//Transport
//----------------------------------------P6015--------------------------------------------------------------
{attribute 'OPC.UA.DA' := '1'}
cfgP6015IntlksArry: ARRAY [0..15] OF ST_CfgEvents := [
   (Description := 'Exit PE/Downstream MTR status' , DeviceLabel := '' , OKState := TRUE),   //DeviceLabel: Exit PE downstream
   (Description := 'System Interlocks' , DeviceLabel := '', OKState := TRUE, StopCode := E_StopCodes.SystemStop),
   (),
   (Description := 'Powered Transfer Raised' , DeviceLabel := 'PX_1281', OKState := TRUE),
   11(())];
{attribute 'OPC.UA.DA' := '1'}
cfgP6015EvntsArry: ARRAY [0..15] OF ST_CfgEvents := [
   (Description := 'Jam Detected', DeviceLabel := '', LatchRequired := TRUE, OKState := FALSE, StopCode := E_StopCodes.ProductJam),   //DeviceLabel: Jam PE
   (),
   (Description := 'Disconnect', DeviceLabel := 'DS6015', OKState := TRUE, StopCode := E_StopCodes.DisconnectState),   //DeviceLabel: Motor Disconnect
   (Description := 'System Fault', DeviceLabel := 'System', OKState := TRUE, FaultWarn:= TRUE, StopCode := E_StopCodes.SystemStop),
   (Description := 'Fire Door Closed', DeviceLabel := 'PE_1231', OKState := TRUE, FaultWarn:= TRUE, StopCode := E_StopCodes.SystemStop),
   (Description := 'RIO1181 Comm Fault', DeviceLabel := 'RIO1181', OKState := TRUE, FaultWarn:= TRUE, StopCode := E_StopCodes.FieldIOFLT),
   (Description := 'Motor Faulted', DeviceLabel := 'P6015', OKState := FALSE, StopCode := E_StopCodes.MotorOL),
   9(())];
//----------------------------------------P6020--------------------------------------------------------------
{attribute 'OPC.UA.DA' := '1'}
cfgP6020IntlksArry: ARRAY [0..15] OF ST_CfgEvents := [
   (Description := 'Exit PE/Downstream MTR status' , DeviceLabel := '' , OKState := TRUE),   //DeviceLabel: Exit PE downstream
   (Description := 'System Interlocks' , DeviceLabel := '', OKState := TRUE, StopCode := E_StopCodes.SystemStop),
   (),
   13(())];
{attribute 'OPC.UA.DA' := '1'}
cfgP6020EvntsArry: ARRAY [0..15] OF ST_CfgEvents := [
   (Description := 'Jam Detected', DeviceLabel := '', LatchRequired := TRUE, OKState := FALSE, StopCode := E_StopCodes.ProductJam),   //DeviceLabel: Jam PE
   (),
   (Description := 'Disconnect', DeviceLabel := 'DS6020', OKState := TRUE, StopCode := E_StopCodes.DisconnectState),   //DeviceLabel: Motor Disconnect
   (Description := 'System Fault', DeviceLabel := 'System', OKState := TRUE, FaultWarn:= TRUE, StopCode := E_StopCodes.SystemStop),
   (Description := 'RIO16171 Comm Fault', DeviceLabel := 'RIO1181', OKState := TRUE, FaultWarn:= TRUE, StopCode := E_StopCodes.FieldIOFLT),
   (Description := 'Motor Faulted', DeviceLabel := 'P6020', OKState := FALSE, StopCode := E_StopCodes.MotorOL),
   10(())];
//----------------------------------------P6025--------------------------------------------------------------
{attribute 'OPC.UA.DA' := '1'}
cfgP6025IntlksArry: ARRAY [0..15] OF ST_CfgEvents := [
   (Description := 'Exit PE/Downstream MTR status' , DeviceLabel := '' , OKState := TRUE),   //DeviceLabel: Exit PE downstream
   (Description := 'System Interlocks' , DeviceLabel := '', OKState := TRUE, StopCode := E_StopCodes.SystemStop),
   (),
   13(())];
{attribute 'OPC.UA.DA' := '1'}
cfgP6025EvntsArry: ARRAY [0..15] OF ST_CfgEvents := [
   (Description := 'Jam Detected', DeviceLabel := '', LatchRequired := TRUE, OKState := FALSE, StopCode := E_StopCodes.ProductJam),   //DeviceLabel: Jam PE
   (),
   (Description := 'Disconnect', DeviceLabel := 'DS6025', OKState := TRUE, StopCode := E_StopCodes.DisconnectState),   //DeviceLabel: Motor Disconnect
   (Description := 'System Fault', DeviceLabel := 'System', OKState := TRUE, FaultWarn:= TRUE, StopCode := E_StopCodes.SystemStop),
   (Description := 'RIO4172 Comm Fault', DeviceLabel := 'RIO4172', OKState := TRUE, FaultWarn:= TRUE, StopCode := E_StopCodes.FieldIOFLT),
   (Description := 'Motor Faulted', DeviceLabel := 'P6025', OKState := FALSE, StopCode := E_StopCodes.MotorOL),
   10(())];
//----------------------------------------P6030--------------------------------------------------------------
{attribute 'OPC.UA.DA' := '1'}
cfgP6030IntlksArry: ARRAY [0..15] OF ST_CfgEvents := [
   (Description := 'Exit PE/Downstream MTR status' , DeviceLabel := '' , OKState := TRUE),   //DeviceLabel: Exit PE downstream
   (Description := 'System Interlocks' , DeviceLabel := '', OKState := TRUE, StopCode := E_StopCodes.SystemStop),
   (),
   12(())];
{attribute 'OPC.UA.DA' := '1'}
cfgP6030EvntsArry: ARRAY [0..15] OF ST_CfgEvents := [
   (Description := 'Jam Detected', DeviceLabel := '', LatchRequired := TRUE, OKState := FALSE, StopCode := E_StopCodes.ProductJam),   //DeviceLabel: Jam PE
   (),
   (Description := 'Disconnect', DeviceLabel := 'DS6030', OKState := TRUE, StopCode := E_StopCodes.DisconnectState),   //DeviceLabel: Motor Disconnect
   (Description := 'System Fault', DeviceLabel := 'System', OKState := TRUE, FaultWarn:= TRUE, StopCode := E_StopCodes.SystemStop),
   (Description := 'RIO4172 Comm Fault', DeviceLabel := 'RIO4172', OKState := TRUE, FaultWarn:= TRUE, StopCode := E_StopCodes.FieldIOFLT),
   (Description := 'Motor Faulted', DeviceLabel := 'P6030', OKState := FALSE, StopCode := E_StopCodes.MotorOL),
   10(())];
//----------------------------------------P6035--------------------------------------------------------------
{attribute 'OPC.UA.DA' := '1'}
cfgP6035IntlksArry: ARRAY [0..15] OF ST_CfgEvents := [
   (Description := 'Exit PE/Downstream MTR status' , DeviceLabel := '' , OKState := TRUE),   //DeviceLabel: Exit PE downstream
   (Description := 'System Interlocks' , DeviceLabel := '', OKState := TRUE, StopCode := E_StopCodes.SystemStop),
   (),
   12(())];
{attribute 'OPC.UA.DA' := '1'}
cfgP6035EvntsArry: ARRAY [0..15] OF ST_CfgEvents := [
   (Description := 'Jam Detected', DeviceLabel := '', LatchRequired := TRUE, OKState := FALSE, StopCode := E_StopCodes.ProductJam),   //DeviceLabel: Jam PE
   (),
   (Description := 'Disconnect', DeviceLabel := 'DS6035', OKState := TRUE, StopCode := E_StopCodes.DisconnectState),   //DeviceLabel: Motor Disconnect
   (Description := 'System Fault', DeviceLabel := 'System', OKState := TRUE, FaultWarn:= TRUE, StopCode := E_StopCodes.SystemStop),
   (Description := 'RIO4172 Comm Fault', DeviceLabel := 'RIO4172', OKState := TRUE, FaultWarn:= TRUE, StopCode := E_StopCodes.FieldIOFLT),
   (Description := 'Motor Faulted', DeviceLabel := 'P6035', OKState := FALSE, StopCode := E_StopCodes.MotorOL),
   10(())];
//Spiral
//----------------------------------------P6045--------------------------------------------------------------
{attribute 'OPC.UA.DA' := '1'}
cfgP6045IntlksArry: ARRAY [0..15] OF ST_CfgEvents := [
   (Description := 'Exit PE/Downstream MTR status' , DeviceLabel := '' , OKState := TRUE),   //DeviceLabel: Exit PE downstream
   (Description := 'System Interlocks' , DeviceLabel := '', OKState := TRUE, StopCode := E_StopCodes.SystemStop),
   (),
   12(())];
{attribute 'OPC.UA.DA' := '1'}
cfgP6045EvntsArry: ARRAY [0..15] OF ST_CfgEvents := [
   (Description := 'Jam Detected', DeviceLabel := '', LatchRequired := TRUE, OKState := FALSE, StopCode := E_StopCodes.ProductJam),   //DeviceLabel: Jam PE
   (),
   (Description := 'Disconnect', DeviceLabel := 'DS6045', OKState := TRUE, StopCode := E_StopCodes.DisconnectState),   //DeviceLabel: Motor Disconnect
   (Description := 'System Fault', DeviceLabel := 'System', OKState := TRUE, FaultWarn:= TRUE, StopCode := E_StopCodes.SystemStop),
   (Description := 'RIO4172 Comm Fault', DeviceLabel := 'RIO4172', OKState := TRUE, FaultWarn:= TRUE, StopCode := E_StopCodes.FieldIOFLT),
   (Description := 'VFD State Not OK', DeviceLabel := 'P6045', OKState := TRUE, StopCode := E_StopCodes.VFD_Fault),
   10(())];
//Sorter
//----------------------------------------P6040--------------------------------------------------------------
{attribute 'OPC.UA.DA' := '1'}
cfgP6040IntlksArry: ARRAY [0..15] OF ST_CfgEvents := [
   (Description := 'Exit PE/Downstream MTR status' , DeviceLabel := '' , OKState := TRUE),   //DeviceLabel: Exit PE downstream
   (Description := 'System Interlocks' , DeviceLabel := '', OKState := TRUE, StopCode := E_StopCodes.SystemStop),
   (Description := 'GR6040-01 Auto', DeviceLabel := 'GR6040-01', OKState := TRUE, StopCode := E_StopCodes.DeviceNoInAuto),
   (Description := 'GR6040-02 Auto', DeviceLabel := 'GR6040-02', OKState := TRUE, StopCode := E_StopCodes.DeviceNoInAuto),
   (Description := 'PI6040-01 Auto', DeviceLabel := 'PI6040-01', OKState := TRUE, StopCode := E_StopCodes.DeviceNoInAuto),
   (Description := 'PU6040-01 Auto', DeviceLabel := 'PU6040-01', OKState := TRUE, StopCode := E_StopCodes.DeviceNoInAuto),
   (Description := 'PU6040-02 Auto', DeviceLabel := 'PU6040-02', OKState := TRUE, StopCode := E_StopCodes.DeviceNoInAuto),
   (Description := 'PU6040-03 Auto', DeviceLabel := 'PU6040-03', OKState := TRUE, StopCode := E_StopCodes.DeviceNoInAuto),
   (Description := 'PU6040-04 Auto', DeviceLabel := 'PU6040-04', OKState := TRUE, StopCode := E_StopCodes.DeviceNoInAuto),
   (Description := 'Motor Faulted', DeviceLabel := 'P6030', OKState := FALSE, StopCode := E_StopCodes.MotorOL),
   6(())];
{attribute 'OPC.UA.DA' := '1'}
cfgP6040EvntsArry: ARRAY [0..15] OF ST_CfgEvents := [
   (Description := 'Jam Detected', DeviceLabel := '', LatchRequired := TRUE, OKState := FALSE, StopCode := E_StopCodes.ProductJam),   //DeviceLabel: Jam PE
   (),
   (Description := 'Disconnect', DeviceLabel := 'DS6040', OKState := TRUE, StopCode := E_StopCodes.DisconnectState),   //DeviceLabel: Motor Disconnect
   (Description := 'System Fault', DeviceLabel := 'System', OKState := TRUE, FaultWarn:= TRUE, StopCode := E_StopCodes.SystemStop),
   (Description := 'RIO6171 Comm Fault', DeviceLabel := 'RIO6171', OKState := TRUE, FaultWarn:= TRUE, StopCode := E_StopCodes.FieldIOFLT),
   (Description := 'RIO7161 Comm Fault', DeviceLabel := 'RIO7161', OKState := TRUE, FaultWarn:= TRUE, StopCode := E_StopCodes.FieldIOFLT),
   (Description := 'RIO8181 Comm Fault', DeviceLabel := 'RIO8081', OKState := TRUE, FaultWarn:= TRUE, StopCode := E_StopCodes.FieldIOFLT),
   (Description := 'Motor Faulted', DeviceLabel := 'P6030', OKState := FALSE, StopCode := E_StopCodes.MotorOL),
   8(())];
//Conveyors Outgoing 7000 (Orange line)
//Loading Zone
//----------------------------------------P7004--------------------------------------------------------------
{attribute 'OPC.UA.DA' := '1'}
cfgP7004IntlksArry: ARRAY [0..15] OF ST_CfgEvents := [
   (Description := 'Exit PE/Downstream MTR status' , DeviceLabel := '' , OKState := TRUE),   //DeviceLabel: Exit PE downstream
   (Description := 'System Interlocks' , DeviceLabel := '', OKState := TRUE, StopCode := E_StopCodes.SystemStop),
   (),
   12(())];
{attribute 'OPC.UA.DA' := '1'}
cfgP7004EvntsArry: ARRAY [0..15] OF ST_CfgEvents := [
   (Description := 'Jam Detected', DeviceLabel := '', LatchRequired := TRUE, OKState := FALSE, StopCode := E_StopCodes.ProductJam),   //DeviceLabel: Jam PE
   (),
   (Description := 'Disconnect', DeviceLabel := 'DS7004', OKState := TRUE, StopCode := E_StopCodes.DisconnectState),   //DeviceLabel: Motor Disconnect
   (Description := 'System Fault', DeviceLabel := 'System', OKState := TRUE, FaultWarn:= TRUE, StopCode := E_StopCodes.SystemStop),
   (Description := 'Height Check', DeviceLabel := 'PE_12261', OKState := TRUE, FaultWarn:= TRUE, StopCode := E_StopCodes.OverHeightFLT),
   (Description := 'RIO12171 Comm Fault', DeviceLabel := 'RIO12171', OKState := TRUE, FaultWarn:= TRUE, StopCode := E_StopCodes.FieldIOFLT),
   (Description := 'Motor Faulted', DeviceLabel := 'P6030', OKState := FALSE, StopCode := E_StopCodes.MotorOL),
   9(())];
//Spiral
//----------------------------------------P7005--------------------------------------------------------------
{attribute 'OPC.UA.DA' := '1'}
cfgP7005IntlksArry: ARRAY [0..15] OF ST_CfgEvents := [
   (Description := 'Exit PE/Downstream MTR status' , DeviceLabel := '' , OKState := TRUE),   //DeviceLabel: Exit PE downstream
   (Description := 'System Interlocks' , DeviceLabel := '', OKState := TRUE, StopCode := E_StopCodes.SystemStop),
   (),
   12(())];
{attribute 'OPC.UA.DA' := '1'}
cfgP7005EvntsArry: ARRAY [0..15] OF ST_CfgEvents := [
   (Description := 'Jam Detected', DeviceLabel := '', LatchRequired := TRUE, OKState := FALSE, StopCode := E_StopCodes.ProductJam),   //DeviceLabel: Jam PE
   (),
   (Description := 'Disconnect', DeviceLabel := 'DS7005', OKState := TRUE, StopCode := E_StopCodes.DisconnectState),   //DeviceLabel: Motor Disconnect
   (Description := 'System Fault', DeviceLabel := 'System', OKState := TRUE, FaultWarn:= TRUE, StopCode := E_StopCodes.SystemStop),
   (Description := 'RIO12171 Comm Fault', DeviceLabel := 'RIO12171', OKState := TRUE, FaultWarn:= TRUE, StopCode := E_StopCodes.FieldIOFLT),
   (Description := 'VFD State Not OK', DeviceLabel := 'P7005', OKState := TRUE, StopCode := E_StopCodes.VFD_Fault),
   10(())];
//Transport
//----------------------------------------P7010--------------------------------------------------------------
{attribute 'OPC.UA.DA' := '1'}
cfgP7010IntlksArry: ARRAY [0..15] OF ST_CfgEvents := [
   (Description := 'Exit PE/Downstream MTR status' , DeviceLabel := '' , OKState := TRUE),   //DeviceLabel: Exit PE downstream
   (Description := 'System Interlocks' , DeviceLabel := '', OKState := TRUE, StopCode := E_StopCodes.SystemStop),
   (),
   12(())];
{attribute 'OPC.UA.DA' := '1'}
cfgP7010EvntsArry: ARRAY [0..15] OF ST_CfgEvents := [
   (Description := 'Jam Detected', DeviceLabel := '', LatchRequired := TRUE, OKState := FALSE, StopCode := E_StopCodes.ProductJam),   //DeviceLabel: Jam PE
   (),
   (Description := 'Disconnect', DeviceLabel := '', OKState := TRUE, StopCode := E_StopCodes.DisconnectState),   //DeviceLabel: Motor Disconnect
   (Description := 'System Fault', DeviceLabel := 'System', OKState := TRUE, FaultWarn:= TRUE, StopCode := E_StopCodes.SystemStop),
   (Description := 'RIO12171 Comm Fault', DeviceLabel := 'RIO12171', OKState := TRUE, FaultWarn:= TRUE, StopCode := E_StopCodes.FieldIOFLT),
   (Description := 'Motor Faulted', DeviceLabel := 'P7010', OKState := FALSE, StopCode := E_StopCodes.MotorOL),
   10(())];
//----------------------------------------P7015--------------------------------------------------------------
{attribute 'OPC.UA.DA' := '1'}
cfgP7015IntlksArry: ARRAY [0..15] OF ST_CfgEvents := [
   (Description := 'Exit PE/Downstream MTR status' , DeviceLabel := '' , OKState := TRUE),   //DeviceLabel: Exit PE downstream
   (Description := 'System Interlocks' , DeviceLabel := '', OKState := TRUE, StopCode := E_StopCodes.SystemStop),
   (),
   12(())];
{attribute 'OPC.UA.DA' := '1'}
cfgP7015EvntsArry: ARRAY [0..15] OF ST_CfgEvents := [
   (Description := 'Jam Detected', DeviceLabel := '', LatchRequired := TRUE, OKState := FALSE, StopCode := E_StopCodes.ProductJam),   //DeviceLabel: Jam PE
   (),
   (Description := 'Disconnect', DeviceLabel := '', OKState := TRUE, StopCode := E_StopCodes.DisconnectState),   //DeviceLabel: Motor Disconnect
   (Description := 'System Fault', DeviceLabel := 'System', OKState := TRUE, FaultWarn:= TRUE, StopCode := E_StopCodes.SystemStop),
   (Description := 'RIO15181 Comm Fault', DeviceLabel := 'RIO15181', OKState := TRUE, FaultWarn:= TRUE, StopCode := E_StopCodes.FieldIOFLT),
   (Description := 'Motor Faulted', DeviceLabel := 'P7015', OKState := FALSE, StopCode := E_StopCodes.MotorOL),
   10(())];
//----------------------------------------P7020--------------------------------------------------------------
{attribute 'OPC.UA.DA' := '1'}
cfgP7020IntlksArry: ARRAY [0..15] OF ST_CfgEvents := [
   (Description := 'Exit PE/Downstream MTR status' , DeviceLabel := '' , OKState := TRUE),   //DeviceLabel: Exit PE downstream
   (Description := 'System Interlocks' , DeviceLabel := '', OKState := TRUE, StopCode := E_StopCodes.SystemStop),
   (),
   12(())];
{attribute 'OPC.UA.DA' := '1'}
cfgP7020EvntsArry: ARRAY [0..15] OF ST_CfgEvents := [
   (Description := 'Jam Detected', DeviceLabel := '', LatchRequired := TRUE, OKState := FALSE, StopCode := E_StopCodes.ProductJam),   //DeviceLabel: Jam PE
   (),
   (Description := 'Disconnect', DeviceLabel := '', OKState := TRUE, StopCode := E_StopCodes.DisconnectState),   //DeviceLabel: Motor Disconnect
   (Description := 'System Fault', DeviceLabel := 'System', OKState := TRUE, FaultWarn:= TRUE, StopCode := E_StopCodes.SystemStop),
   (Description := 'RIO15181 Comm Fault', DeviceLabel := 'RIO15181', OKState := TRUE, FaultWarn:= TRUE, StopCode := E_StopCodes.FieldIOFLT),
   (Description := 'Motor Faulted', DeviceLabel := 'P7020', OKState := FALSE, StopCode := E_StopCodes.MotorRunTO),
   10(())];
//----------------------------------------P7025--------------------------------------------------------------
{attribute 'OPC.UA.DA' := '1'}
cfgP7025IntlksArry: ARRAY [0..15] OF ST_CfgEvents := [
   (Description := 'Exit PE/Downstream MTR status' , DeviceLabel := '' , OKState := TRUE),   //DeviceLabel: Exit PE downstream
   (Description := 'System Interlocks' , DeviceLabel := '', OKState := TRUE, StopCode := E_StopCodes.SystemStop),
   (),
   12(())];
{attribute 'OPC.UA.DA' := '1'}
cfgP7025EvntsArry: ARRAY [0..15] OF ST_CfgEvents := [
   (Description := 'Jam Detected', DeviceLabel := '', LatchRequired := TRUE, OKState := FALSE, StopCode := E_StopCodes.ProductJam),   //DeviceLabel: Jam PE
   (),
   (Description := 'Disconnect', DeviceLabel := '', OKState := TRUE, StopCode := E_StopCodes.DisconnectState),   //DeviceLabel: Motor Disconnect
   (Description := 'System Fault', DeviceLabel := 'System', OKState := TRUE, FaultWarn:= TRUE, StopCode := E_StopCodes.SystemStop),
   (Description := 'RIO15181 Comm Fault', DeviceLabel := 'RIO15181', OKState := TRUE, FaultWarn:= TRUE, StopCode := E_StopCodes.FieldIOFLT),
   (Description := 'Motor Faulted', DeviceLabel := 'P7025', OKState := FALSE, StopCode := E_StopCodes.MotorOL),
   10(())];
//----------------------------------------P7030--------------------------------------------------------------
{attribute 'OPC.UA.DA' := '1'}
cfgP7030IntlksArry: ARRAY [0..15] OF ST_CfgEvents := [
   (Description := 'Exit PE/Downstream MTR status' , DeviceLabel := '' , OKState := TRUE),   //DeviceLabel: Exit PE downstream
   (Description := 'System Interlocks' , DeviceLabel := '', OKState := TRUE, StopCode := E_StopCodes.SystemStop),
   (),
   12(())];
{attribute 'OPC.UA.DA' := '1'}
cfgP7030EvntsArry: ARRAY [0..15] OF ST_CfgEvents := [
   (Description := 'Jam Detected', DeviceLabel := '', LatchRequired := TRUE, OKState := FALSE, StopCode := E_StopCodes.ProductJam),   //DeviceLabel: Jam PE
   (),
   (Description := 'Disconnect', DeviceLabel := '', OKState := TRUE, StopCode := E_StopCodes.DisconnectState),   //DeviceLabel: Motor Disconnect
   (Description := 'System Fault', DeviceLabel := 'System', OKState := TRUE, FaultWarn:= TRUE, StopCode := E_StopCodes.SystemStop),
   (Description := 'RIO16171 Comm Fault', DeviceLabel := 'RIO16171', OKState := TRUE, FaultWarn:= TRUE, StopCode := E_StopCodes.FieldIOFLT),
   (Description := 'Motor Faulted', DeviceLabel := 'P7030', OKState := FALSE, StopCode := E_StopCodes.MotorOL),
   10(())];
//----------------------------------------P7035--------------------------------------------------------------
{attribute 'OPC.UA.DA' := '1'}
cfgP7035IntlksArry: ARRAY [0..15] OF ST_CfgEvents := [
   (Description := 'Exit PE/Downstream MTR status' , DeviceLabel := '' , OKState := TRUE),   //DeviceLabel: Exit PE downstream
   (Description := 'System Interlocks' , DeviceLabel := '', OKState := TRUE, StopCode := E_StopCodes.SystemStop),
   (),
   (Description := 'Powered Transfer Raised' , DeviceLabel := 'PX_16231', OKState := TRUE),
   12(())];
{attribute 'OPC.UA.DA' := '1'}
cfgP7035EvntsArry: ARRAY [0..15] OF ST_CfgEvents := [
   (Description := 'Jam Detected', DeviceLabel := '', LatchRequired := TRUE, OKState := FALSE, StopCode := E_StopCodes.ProductJam),   //DeviceLabel: Jam PE
   (),
   (Description := 'Disconnect', DeviceLabel := '', OKState := TRUE, StopCode := E_StopCodes.DisconnectState),   //DeviceLabel: Motor Disconnect
   (Description := 'System Fault', DeviceLabel := 'System', OKState := TRUE, FaultWarn:= TRUE, StopCode := E_StopCodes.SystemStop),
   (Description := 'Fire Door Closed', DeviceLabel := 'PE_16181', OKState := TRUE, FaultWarn:= TRUE, StopCode := E_StopCodes.SystemStop),
   (Description := 'RIO16171 Comm Fault', DeviceLabel := 'RIO16171', OKState := TRUE, FaultWarn:= TRUE, StopCode := E_StopCodes.FieldIOFLT),
   (Description := 'Motor Faulted', DeviceLabel := 'P7035', OKState := FALSE, StopCode := E_StopCodes.MotorOL),
   9(())];
//Spiral
//----------------------------------------P7040--------------------------------------------------------------
{attribute 'OPC.UA.DA' := '1'}
cfgP7040IntlksArry: ARRAY [0..15] OF ST_CfgEvents := [
   (Description := 'Exit PE/Downstream MTR status' , DeviceLabel := '' , OKState := TRUE),   //DeviceLabel: Exit PE downstream
   (Description := 'System Interlocks' , DeviceLabel := '', OKState := TRUE, StopCode := E_StopCodes.SystemStop),
   (),
   13(())];
{attribute 'OPC.UA.DA' := '1'}
cfgP7040EvntsArry: ARRAY [0..15] OF ST_CfgEvents := [
   (Description := 'Jam Detected', DeviceLabel := '', LatchRequired := TRUE, OKState := FALSE, StopCode := E_StopCodes.ProductJam),   //DeviceLabel: Jam PE
   (),
   (Description := 'Disconnect', DeviceLabel := '', OKState := TRUE, StopCode := E_StopCodes.DisconnectState),   //DeviceLabel: Motor Disconnect
   (Description := 'System Fault', DeviceLabel := 'System', OKState := TRUE, FaultWarn:= TRUE, StopCode := E_StopCodes.SystemStop),
   (Description := 'RIO16171 Comm Fault', DeviceLabel := 'RIO16171', OKState := TRUE, FaultWarn:= TRUE, StopCode := E_StopCodes.FieldIOFLT),
   (Description := 'VFD State Not OK', DeviceLabel := 'P7040', OKState := TRUE, StopCode := E_StopCodes.VFD_Fault),
   10(())];

//Transport
//----------------------------------------P7045--------------------------------------------------------------
{attribute 'OPC.UA.DA' := '1'}
cfgP7045IntlksArry: ARRAY [0..15] OF ST_CfgEvents := [
   (Description := 'Exit PE/Downstream MTR status' , DeviceLabel := '' , OKState := TRUE),   //DeviceLabel: Exit PE downstream
   (Description := 'System Interlocks' , DeviceLabel := '', OKState := TRUE, StopCode := E_StopCodes.SystemStop),
   (),
   13(())];
{attribute 'OPC.UA.DA' := '1'}
cfgP7045EvntsArry: ARRAY [0..15] OF ST_CfgEvents := [
   (Description := 'Jam Detected', DeviceLabel := '', LatchRequired := TRUE, OKState := FALSE, StopCode := E_StopCodes.ProductJam),   //DeviceLabel: Jam PE
   (),
   (Description := 'Disconnect', DeviceLabel := '', OKState := TRUE, StopCode := E_StopCodes.DisconnectState),   //DeviceLabel: Motor Disconnect
   (Description := 'System Fault', DeviceLabel := 'System', OKState := TRUE, FaultWarn:= TRUE, StopCode := E_StopCodes.SystemStop),
   (Description := 'Fire Door Closed', DeviceLabel := 'PE_16181', OKState := TRUE, FaultWarn:= TRUE, StopCode := E_StopCodes.SystemStop),
   (Description := 'RIO16171 Comm Fault', DeviceLabel := 'RIO16171', OKState := TRUE, FaultWarn:= TRUE, StopCode := E_StopCodes.FieldIOFLT),
   (Description := 'Motor Faulted', DeviceLabel := 'P7045', OKState := FALSE, StopCode := E_StopCodes.MotorOL),
   9(())];			
END_VAR

ResetAllDrives:=System.Cnvyr_Reset;

//----------------------------------------P6005--------------------------------------------------------------
P6005_StatePB.AutoPB := System.Cnvyr_Auto;
P6005_StatePB.ManPB := System.Cnvyr_Manual;
P6005_StatePB.ResetPB := System.Cnvyr_Reset;
P6005_StatePB.OfflinePB := System.Cnvyr_Offline;
P6005SleepWakeTrig[1] := PhotoEyes.PE_1232.Out;
P6005SleepWakeTrig[2] := GVL_IO.From205_P3130_SendingProduct;		// Belive this will be an EAP photoeye from 3rd floor

GVL_IO.To205_P6005_IsRunning:= P6005_Status.Sts_IsRunning;

// Initialize the Equipment Type
P6005_Status.Sts_EquipmentState.EquipType := E_EquipType.Conveyor;

// Interlocks
//P6005.In_EquipIntlks.2:=  

//Events
  P6005.In_EquipEvents.2:= GVL_IO.DS_P6005;
  P6005.In_EquipEvents.3:= System.SysEventsAllOk;
  P6005.In_EquipEvents.4:= Photoeyes.PE_1231.Out; //Goes low when door drops
  P6005.In_EquipEvents.5:= NOT CommStatus.RIO1181_CommFault.Out;
  P6005.In_EquipEvents.6:= NOT GVL_IO.P6005_Faulted;

// Function Call
P6005(
   In_p_EquipStatePB:= P6005_StatePB,
   In_P_ConvReqRun:= TRUE,
   In_ConvDwnStrmMtrStatus:= P6010_VFD.IsRunning,
   In_ConvCrntExitPhotoEye:= Photoeyes.PE_1232.Out,
   In_SimActive:= System.Sys_SimActive,
   In_EquipInit:= GVL_IO.INIT,
   In_WakeSlpTrigArry:= P6005SleepWakeTrig,
   Cfg_EquipIndex := GVL_EquipArrays.nEquipIndex,
   Cfg_EquipLabel := cfgP6005Label,
   Cfg_EquipDefState:= System.ConvDefaultState,
   Cfg_EquipIntlksArry:= cfgP6005IntlksArry,
   Cfg_EquipEvntsArry:= cfgP6005EvntsArry,
   cfg_JamDetectTime:= cfgP6005JamDetectTime,
   Cfg_UseSleepTmr := TRUE,
   Cfg_UseStartUpDelay := TRUE,
   Cfg_StartUpDelayTime := T#500MS,
   Cfg_SleepWaitTime:= cfgP6005SleepTime,
   Sts_EquipState := P6005_Status,
   Out_ConvCrntMtr => GVL_IO.P6005_RUN);

P6005_Status.Sts_IsRunning := GVL_IO.P6005_RUN;
//----------------------------------------P6010--------------------------------------------------------------
P6010_StatePB.AutoPB := System.Cnvyr_Auto;
P6010_StatePB.ManPB := System.Cnvyr_Manual;
P6010_StatePB.ResetPB := System.Cnvyr_Reset;
P6010_StatePB.OfflinePB := System.Cnvyr_Offline;
P6010SleepWakeTrig[1] := PhotoEyes.PE_1232.Out_OffFltrd;
P6010SleepWakeTrig[5] := P6005SleepWakeTrig[1]
						OR P6005SleepWakeTrig[2]
						OR P6005SleepWakeTrig[3]
						OR P6005SleepWakeTrig[4]
						OR P6005SleepWakeTrig[5];
// ADD an EAP photoeye from 3rd floor

// Initialize the Equipment Type
P6010_Status.Sts_EquipmentState.EquipType := E_EquipType.Conveyor;

// Interlocks
 // P6010.In_EquipIntlks.2:= 
//Events
  P6010.In_EquipEvents.2:= GVL_IO.DS_P6010;
  P6010.In_EquipEvents.3:= System.SysEventsAllOk;
  P6010.In_EquipEvents.4:= NOT CommStatus.RIO1181_CommFault.Out;
  P6010.In_EquipEvents.5:= NOT P6010_VFD.IsFaulted;

// Function Call
P6010(
   In_p_EquipStatePB:= P6010_StatePB,
   In_P_ConvReqRun:= TRUE,
   In_ConvDwnStrmMtrStatus:= P6015_Status.Sts_IsRunning,
   In_ConvCrntExitPhotoEye:= Photoeyes.PE_1162.Out,
   In_SimActive:= System.Sys_SimActive,
   In_EquipInit:= GVL_IO.INIT,
   In_WakeSlpTrigArry:= P6010SleepWakeTrig,
   Cfg_EquipIndex := GVL_EquipArrays.nEquipIndex,
   Cfg_EquipLabel := cfgP6010Label,
   Cfg_EquipDefState:= System.ConvDefaultState,
   Cfg_EquipIntlksArry:= cfgP6010IntlksArry,
   Cfg_EquipEvntsArry:= cfgP6010EvntsArry,
   cfg_JamDetectTime:= cfgP6010JamDetectTime,
   Cfg_UseSleepTmr := TRUE,
   Cfg_UseStartUpDelay := TRUE,
   Cfg_StartUpDelayTime := T#500MS,
   Cfg_SleepWaitTime:= cfgP6010SleepTime,
   Sts_EquipState := P6010_Status);

//Motor Control
P6010_VFD(
   RunVelocity := DefaultVelocity,
   VelocityThreshold := DefaultVelocityThreshold,
   Reset := ResetAllDrives,
   RunRequest := (P6010.Out_ConvCrntMtr OR Test_VFD_P6010));
P6010_Status.Sts_IsRunning := P6010_VFD.IsRunning;

//----------------------------------------P6015--------------------------------------------------------------
P6015_StatePB.AutoPB := System.Cnvyr_Auto;
P6015_StatePB.ManPB := System.Cnvyr_Manual;
P6015_StatePB.ResetPB := System.Cnvyr_Reset;
P6015_StatePB.OfflinePB := System.Cnvyr_Offline;
P6015SleepWakeTrig[1] := PhotoEyes.PE_1162.Out_OffFltrd;
P6015SleepWakeTrig[2] :=  PhotoEyes.PE_1232.Out_OffFltrd;

// Initialize the Equipment Type
P6015_Status.Sts_EquipmentState.EquipType := E_EquipType.Conveyor;

// Interlocks
  P6015.In_EquipIntlks.3:= ProxSensors.PX_1281_Extended.Out; //Powered Transfer Raised 
//Events
  P6015.In_EquipEvents.2:= GVL_IO.DS_P6015;
  P6015.In_EquipEvents.3:= System.SysEventsAllOk;
  P6015.In_EquipEvents.4:= Photoeyes.PE_1231.Out; //Goes low when door drops
  P6015.In_EquipEvents.5:= NOT CommStatus.RIO1181_CommFault.Out;
  P6015.In_EquipEvents.6:= NOT GVL_IO.P6015_Faulted;

// Function Call
P6015(
   In_p_EquipStatePB:= P6015_StatePB,
   In_P_ConvReqRun:= TRUE,
   In_ConvDwnStrmMtrStatus:= P6020_Status.Sts_IsRunning,
   In_ConvCrntExitPhotoEye:= Photoeyes.PE_1081.Out,
   In_SimActive:= System.Sys_SimActive,
   In_EquipInit:= GVL_IO.INIT,
   In_WakeSlpTrigArry:= P6015SleepWakeTrig,
   Cfg_EquipIndex := GVL_EquipArrays.nEquipIndex,
   Cfg_EquipLabel := cfgP6015Label,
   Cfg_EquipDefState:= System.ConvDefaultState,
   Cfg_EquipIntlksArry:= cfgP6015IntlksArry,
   Cfg_EquipEvntsArry:= cfgP6015EvntsArry,
   cfg_JamDetectTime:= cfgP6015JamDetectTime,
   Cfg_UseSleepTmr := TRUE,
   Cfg_UseStartUpDelay := TRUE,
   Cfg_StartUpDelayTime := T#500MS,
   Cfg_SleepWaitTime:= cfgP6015SleepTime,
   Sts_EquipState := P6015_Status,
   Out_ConvCrntMtr => GVL_IO.P6015_RUN);

P6015_Status.Sts_IsRunning := GVL_IO.P6015_RUN;
//----------------------------------------P6020--------------------------------------------------------------
P6020_StatePB.AutoPB := System.Cnvyr_Auto;
P6020_StatePB.ManPB := System.Cnvyr_Manual;
P6020_StatePB.ResetPB := System.Cnvyr_Reset;
P6020_StatePB.OfflinePB := System.Cnvyr_Offline;
P6020SleepWakeTrig[1] := PhotoEyes.PE_1081.Out_OffFltrd;
P6020SleepWakeTrig[2] := PhotoEyes.PE_1162.Out_OffFltrd;

// Initialize the Equipment Type
P6020_Status.Sts_EquipmentState.EquipType := E_EquipType.Conveyor;

// Interlocks
 // P6020.In_EquipIntlks.2:=
//Events
  P6020.In_EquipEvents.2:= GVL_IO.DS_P6020;
  P6020.In_EquipEvents.3:= System.SysEventsAllOk;
  P6020.In_EquipEvents.4:= NOT CommStatus.RIO1181_CommFault.Out;
  P6020.In_EquipEvents.5:= NOT GVL_IO.P6020_Faulted;

// Function Call
P6020(
   In_p_EquipStatePB:= P6020_StatePB,
   In_P_ConvReqRun:= TRUE,
   In_ConvDwnStrmMtrStatus:= P6025_Status.Sts_IsRunning,
   In_ConvCrntExitPhotoEye:= Photoeyes.PE_1161.Out,
   In_SimActive:= System.Sys_SimActive,
   In_EquipInit:= GVL_IO.INIT,
   In_WakeSlpTrigArry:= P6020SleepWakeTrig,
   Cfg_EquipIndex := GVL_EquipArrays.nEquipIndex,
   Cfg_EquipLabel := cfgP6020Label,
   Cfg_EquipDefState:= System.ConvDefaultState,
   Cfg_EquipIntlksArry:= cfgP6020IntlksArry,
   Cfg_EquipEvntsArry:= cfgP6020EvntsArry,
   cfg_JamDetectTime:= cfgP6020JamDetectTime,
   Cfg_UseSleepTmr := TRUE,
   Cfg_UseStartUpDelay := TRUE,
   Cfg_StartUpDelayTime := T#500MS,
   Cfg_SleepWaitTime:= cfgP6020SleepTime,
   Sts_EquipState := P6020_Status,
   Out_ConvCrntMtr => GVL_IO.P6020_RUN);

P6020_Status.Sts_IsRunning := GVL_IO.P6020_RUN;
//----------------------------------------P6025--------------------------------------------------------------
P6025_StatePB.AutoPB := System.Cnvyr_Auto;
P6025_StatePB.ManPB := System.Cnvyr_Manual;
P6025_StatePB.ResetPB := System.Cnvyr_Reset;
P6025_StatePB.OfflinePB := System.Cnvyr_Offline;
P6025SleepWakeTrig[1] := PhotoEyes.PE_1161.Out_OffFltrd;
P6025SleepWakeTrig[2] := PhotoEyes.PE_1081.Out_OffFltrd;

// Initialize the Equipment Type
P6025_Status.Sts_EquipmentState.EquipType := E_EquipType.Conveyor;

// Interlocks
//  P6025.In_EquipIntlks.2:= 
//Events
  P6025.In_EquipEvents.2:= GVL_IO.DS_P6025;
  P6025.In_EquipEvents.3:= System.SysEventsAllOk;
  P6025.In_EquipEvents.4:= NOT CommStatus.RIO4172_CommFault.Out;
  P6025.In_EquipEvents.5:= NOT GVL_IO.P6025_Faulted;

// Function Call
P6025(
   In_p_EquipStatePB:= P6025_StatePB,
   In_P_ConvReqRun:= TRUE,
   In_ConvDwnStrmMtrStatus:= P6030_Status.Sts_IsRunning,
   In_ConvCrntExitPhotoEye:= Photoeyes.PE_4121.Out,
   In_SimActive:= System.Sys_SimActive,
   In_EquipInit:= GVL_IO.INIT,
   In_WakeSlpTrigArry:= P6025SleepWakeTrig,
   Cfg_EquipIndex := GVL_EquipArrays.nEquipIndex,
   Cfg_EquipLabel := cfgP6025Label,
   Cfg_EquipDefState:= System.ConvDefaultState,
   Cfg_EquipIntlksArry:= cfgP6025IntlksArry,
   Cfg_EquipEvntsArry:= cfgP6025EvntsArry,
   cfg_JamDetectTime:= cfgP6025JamDetectTime,
   Cfg_UseSleepTmr := TRUE,
   Cfg_UseStartUpDelay := TRUE,
   Cfg_StartUpDelayTime := T#500MS,
   Cfg_SleepWaitTime:= cfgP6025SleepTime,
   Sts_EquipState := P6025_Status,
   Out_ConvCrntMtr => GVL_IO.P6025_RUN);

P6025_Status.Sts_IsRunning := GVL_IO.P6025_RUN;
//----------------------------------------P6030--------------------------------------------------------------
P6030_StatePB.AutoPB := System.Cnvyr_Auto;
P6030_StatePB.ManPB := System.Cnvyr_Manual;
P6030_StatePB.ResetPB := System.Cnvyr_Reset;
P6030_StatePB.OfflinePB := System.Cnvyr_Offline;
P6030SleepWakeTrig[1] := PhotoEyes.PE_4121.Out_OffFltrd;
P6030SleepWakeTrig[2] := PhotoEyes.PE_1161.Out_OffFltrd;

// Initialize the Equipment Type
P6030_Status.Sts_EquipmentState.EquipType := E_EquipType.Conveyor;

// Interlocks
// P6030.In_EquipIntlks.2:= 
//Events
  P6030.In_EquipEvents.2:= GVL_IO.DS_P6030;
  P6030.In_EquipEvents.3:= System.SysEventsAllOk;
  P6030.In_EquipEvents.4:= NOT CommStatus.RIO4172_CommFault.Out;
  P6030.In_EquipEvents.5:= NOT GVL_IO.P6030_Faulted;

// Function Call
P6030(
   In_p_EquipStatePB:= P6030_StatePB,
   In_P_ConvReqRun:= TRUE,
   In_ConvDwnStrmMtrStatus:= P6035_Status.Sts_IsRunning,
   In_ConvCrntExitPhotoEye:= Photoeyes.PE_4271.Out,
   In_SimActive:= System.Sys_SimActive,
   In_EquipInit:= GVL_IO.INIT,
   In_WakeSlpTrigArry:= P6030SleepWakeTrig,
   Cfg_EquipIndex := GVL_EquipArrays.nEquipIndex,
   Cfg_EquipLabel := cfgP6030Label,
   Cfg_EquipDefState:= System.ConvDefaultState,
   Cfg_EquipIntlksArry:= cfgP6030IntlksArry,
   Cfg_EquipEvntsArry:= cfgP6030EvntsArry,
   cfg_JamDetectTime:= cfgP6030JamDetectTime,
   Cfg_UseSleepTmr := TRUE,
   Cfg_UseStartUpDelay := TRUE,
   Cfg_StartUpDelayTime := T#500MS,
   Cfg_SleepWaitTime:= cfgP6030SleepTime,
   Sts_EquipState := P6030_Status,
   Out_ConvCrntMtr => GVL_IO.P6030_RUN);

P6030_Status.Sts_IsRunning := GVL_IO.P6030_RUN;
//----------------------------------------P6035--------------------------------------------------------------
P6035_StatePB.AutoPB := System.Cnvyr_Auto;
P6035_StatePB.ManPB := System.Cnvyr_Manual;
P6035_StatePB.ResetPB := System.Cnvyr_Reset;
P6035_StatePB.OfflinePB := System.Cnvyr_Offline;
P6035SleepWakeTrig[1] := PhotoEyes.PE_4271.Out_OffFltrd;
P6035SleepWakeTrig[2] := PhotoEyes.PE_4121.Out_OffFltrd;

// Initialize the Equipment Type
P6035_Status.Sts_EquipmentState.EquipType := E_EquipType.Conveyor;

// Interlocks
//  P6035.In_EquipIntlks.2:= 
//Events
  P6035.In_EquipEvents.2:= GVL_IO.DS_P6005;
  P6035.In_EquipEvents.3:= System.SysEventsAllOk;
  P6035.In_EquipEvents.4:= NOT CommStatus.RIO4172_CommFault.Out;
  P6035.In_EquipEvents.5:= NOT GVL_IO.P6035_Faulted;
// Function Call
P6035(
   In_p_EquipStatePB:= P6035_StatePB,
   In_P_ConvReqRun:= TRUE,
   In_ConvDwnStrmMtrStatus:= P6045_VFD.IsRunning,
   In_ConvCrntExitPhotoEye:= Photoeyes.PE_4201.Out,
   In_SimActive:= System.Sys_SimActive,
   In_EquipInit:= GVL_IO.INIT,
   In_WakeSlpTrigArry:= P6035SleepWakeTrig,
   Cfg_EquipIndex := GVL_EquipArrays.nEquipIndex,
   Cfg_EquipLabel := cfgP6035Label,
   Cfg_EquipDefState:= System.ConvDefaultState,
   Cfg_EquipIntlksArry:= cfgP6035IntlksArry,
   Cfg_EquipEvntsArry:= cfgP6035EvntsArry,
   cfg_JamDetectTime:= cfgP6035JamDetectTime,
   Cfg_UseSleepTmr := TRUE,
   Cfg_UseStartUpDelay := TRUE,
   Cfg_StartUpDelayTime := T#500MS,
   Cfg_SleepWaitTime:= cfgP6035SleepTime,
   Sts_EquipState := P6035_Status,
   Out_ConvCrntMtr => GVL_IO.P6035_RUN);

P6035_Status.Sts_IsRunning := GVL_IO.P6035_RUN;
//----------------------------------------P6045--------------------------------------------------------------
P6045_StatePB.AutoPB := System.Cnvyr_Auto;
P6045_StatePB.ManPB := System.Cnvyr_Manual;
P6045_StatePB.ResetPB := System.Cnvyr_Reset;
P6045_StatePB.OfflinePB := System.Cnvyr_Offline;
P6045SleepWakeTrig[1] := PhotoEyes.PE_4201.Out_OffFltrd;
P6045SleepWakeTrig[2] := PhotoEyes.PE_4271.Out_OffFltrd;

// Initialize the Equipment Type
P6045_Status.Sts_EquipmentState.EquipType := E_EquipType.Conveyor;

// Interlocks
 P6045.In_EquipIntlks.2:= PhotoEyes.PE_6302.Out;

//Events
  P6045.In_EquipEvents.2:= GVL_IO.DS_P6045;
  P6045.In_EquipEvents.3:= System.SysEventsAllOk;
  P6045.In_EquipEvents.4:= NOT CommStatus.RIO4172_CommFault.Out;
  P6045.In_EquipEvents.5:= NOT P6045_VFD.IsFaulted;

// Function Call
P6045(
   In_p_EquipStatePB:= P6045_StatePB,
   In_P_ConvReqRun:= TRUE,
   In_ConvDwnStrmMtrStatus:= TRUE, //P6040_Status.Sts_IsRunning,
   In_ConvCrntExitPhotoEye:= PhotoEyes.PE_8211.Out,
   In_SimActive:= System.Sys_SimActive,
   In_EquipInit:= GVL_IO.INIT,
   In_WakeSlpTrigArry:= P6045SleepWakeTrig,
   Cfg_EquipIndex := GVL_EquipArrays.nEquipIndex,
   Cfg_EquipLabel := cfgP6045Label,
   Cfg_EquipDefState:= System.ConvDefaultState,
   Cfg_EquipIntlksArry:= cfgP6045IntlksArry,
   Cfg_EquipEvntsArry:= cfgP6045EvntsArry,
   cfg_JamDetectTime:= cfgP6045JamDetectTime,
   Cfg_UseSleepTmr := TRUE,
   Cfg_UseStartUpDelay := FALSE,
   Cfg_SleepWaitTime:= cfgP6045SleepTime,
   Sts_EquipState := P6045_Status);

//Motor Control
P6045_VFD(
   RunVelocity := DefaultVelocity,
   VelocityThreshold := DefaultVelocityThreshold,
   Reset := ResetAllDrives,
   RunRequest := (P6045.Out_ConvCrntMtr OR Test_VFD_P6045));
P6045_Status.Sts_IsRunning := P6045_VFD.IsRunning;
//----------------------------------------P6040--------------------------------------------------------------
P6040_StatePB.AutoPB := System.Cnvyr_Auto;
P6040_StatePB.ManPB := System.Cnvyr_Manual;
P6040_StatePB.ResetPB := System.Cnvyr_Reset;
P6040_StatePB.OfflinePB := System.Cnvyr_Offline;
P6040SleepWakeTrig[1] := PhotoEyes.PE_1162.Out_OffFltrd;
P6040SleepWakeTrig[2] := PhotoEyes.PE_4201.Out_OffFltrd;
P6040SleepWakeTrig[3] := PhotoEyes.PE_6201.Out_OffFltrd;
P6040SleepWakeTrig[4] := PhotoEyes.PE_7171.Out_OffFltrd;
P6040SleepWakeTrig[5] := PhotoEyes.PE_4071.Out_OffFltrd;


// Initialize the Equipment Type
P6040_Status.Sts_EquipmentState.EquipType := E_EquipType.Conveyor;

// Interlocks
P6040.In_EquipIntlks.2:= Solenoids.GR6040_01_Status.Sts_EquipmentState.StsAuto;
P6040.In_EquipIntlks.3:= Solenoids.GR6040_02_Status.Sts_EquipmentState.StsAuto;
P6040.In_EquipIntlks.4:= Solenoids.PI6040_01_Status.Sts_EquipmentState.StsAuto;
P6040.In_EquipIntlks.5:= Solenoids.PU6040_01_Status.Sts_EquipmentState.StsAuto;
P6040.In_EquipIntlks.6:= Solenoids.PU6040_02_Status.Sts_EquipmentState.StsAuto;
P6040.In_EquipIntlks.7:= Solenoids.PU6040_03_Status.Sts_EquipmentState.StsAuto;
P6040.In_EquipIntlks.8:= Solenoids.PU6040_04_Status.Sts_EquipmentState.StsAuto;


//Events
P6040.In_EquipEvents.2:= GVL_IO.DS_P6040;
P6040.In_EquipEvents.3:= System.SysEventsAllOk;
P6040.In_EquipEvents.4:= NOT CommStatus.RIO6171_CommFault.Out;
P6040.In_EquipEvents.5:= NOT CommStatus.RIO7161_CommFault.Out;
P6040.In_EquipEvents.6:= NOT CommStatus.RIO8181_CommFault.Out;
P6040.In_EquipEvents.7:= NOT GVL_IO.P6040_Faulted; 


// Function Call
P6040(
   In_p_EquipStatePB:= P6040_StatePB,
   In_P_ConvReqRun:= TRUE,
   In_ConvDwnStrmMtrStatus:= TRUE,
   In_ConvCrntExitPhotoEye:= PhotoEyes.PE_8211.Out,
   Cfg_ConvType:= E_ConvType.end,
   In_SimActive:= System.Sys_SimActive,
   In_EquipInit:= GVL_IO.INIT,
   In_WakeSlpTrigArry:= P6040SleepWakeTrig,
   Cfg_EquipIndex := GVL_EquipArrays.nEquipIndex,
   Cfg_EquipLabel := cfgP6040Label,
   Cfg_EquipDefState:= System.ConvDefaultState,
   Cfg_EquipIntlksArry:= cfgP6040IntlksArry,
   Cfg_EquipEvntsArry:= cfgP6040EvntsArry,
   cfg_JamDetectTime:= cfgP6040JamDetectTime,
   Cfg_UseSleepTmr := TRUE,
   Cfg_SleepWaitTime:= cfgP6040SleepTime,
   Sts_EquipState := P6040_Status,
   Out_ConvCrntMtr => GVL_IO.P6040_RUN);

P6040_Status.Sts_IsRunning := GVL_IO.P6040_RUN;
//----------------------------------------P7004--------------------------------------------------------------
P7004_StatePB.AutoPB := System.Cnvyr_Auto OR GVL_IO.PB_RemoteReset_12181;
P7004_StatePB.ManPB := System.Cnvyr_Manual;
P7004_StatePB.ResetPB := System.Cnvyr_Reset OR GVL_IO.PB_RemoteReset_12181;
P7004_StatePB.OfflinePB := System.Cnvyr_Offline;
P7004SleepWakeTrig[1] := TRUE; //This conveyor doesn't sleep

// Initialize the Equipment Type
P7004_Status.Sts_EquipmentState.EquipType := E_EquipType.Conveyor;

// Interlocks
  P7004.In_EquipIntlks.2:= FALSE;
//Events
 P7004.In_EquipEvents.2:= GVL_IO.DS_P7004;
 P7004.In_EquipEvents.3:= System.SysEventsAllOk;
 P7004.In_EquipEvents.4:= PhotoEyes.PE_12261.Out;
 P7004.In_EquipEvents.5:= NOT CommStatus.RIO12171_CommFault.Out;
 P7004.In_EquipEvents.6:= NOT GVL_IO.P7004_Faulted;

// Function Call
P7004(
   In_p_EquipStatePB:= P7004_StatePB,
   In_P_ConvReqRun:= TRUE,
   In_ConvDwnStrmMtrStatus:= P7005_VFD.IsRunning,
   In_ConvCrntExitPhotoEye:= FALSE, 
   Cfg_ConvType:= E_ConvType.slave,
   In_SimActive:= System.Sys_SimActive,
   In_EquipInit:= GVL_IO.INIT,
   In_WakeSlpTrigArry:= P7004SleepWakeTrig,
   Cfg_EquipIndex := GVL_EquipArrays.nEquipIndex,
   Cfg_EquipLabel := cfgP7004Label,
   Cfg_EquipDefState:= System.ConvDefaultState,
   Cfg_EquipIntlksArry:= cfgP7004IntlksArry,
   Cfg_EquipEvntsArry:= cfgP7004EvntsArry,
   cfg_JamDetectTime:= cfgP7004JamDetectTime,
   Cfg_UseSleepTmr := TRUE,
   Cfg_UseStartUpDelay := TRUE,
   Cfg_StartUpDelayTime := T#500MS,
   Cfg_SleepWaitTime:= cfgP7004SleepTime,
   Sts_EquipState := P7004_Status,
   Out_ConvCrntMtr => GVL_IO.P7004_RUN);

P7004_Status.Sts_IsRunning := GVL_IO.P7004_RUN;
//----------------------------------------P7005--------------------------------------------------------------
P7005_StatePB.AutoPB := System.Cnvyr_Auto OR GVL_IO.PB_RemoteReset_12181;
P7005_StatePB.ManPB := System.Cnvyr_Manual;
P7005_StatePB.ResetPB := System.Cnvyr_Reset OR GVL_IO.PB_RemoteReset_12181;
P7005_StatePB.OfflinePB := System.Cnvyr_Offline;
P7005_ResetWakeTmr(IN:= GVL_IO.PB_RemoteReset_12181, PT:= T#3S, Q=> );
P7005SleepWakeTrig[1] := PhotoEyes.PE_12221.Out_OffFltrd;
P7005SleepWakeTrig[2] := P7005_ResetWakeTmr.Q; //RESET BUTTON

// Initialize the Equipment Type
P7005_Status.Sts_EquipmentState.EquipType := E_EquipType.Conveyor;

// Interlocks
  P7005.In_EquipIntlks.2:= FALSE;
//Events
  P7005.In_EquipEvents.2:= GVL_IO.DS_P7005;
  P7005.In_EquipEvents.3:= System.SysEventsAllOk;
  P7005.In_EquipEvents.4:= NOT CommStatus.RIO12171_CommFault.Out;
  P7005.In_EquipEvents.5:= PhotoEyes.PE_12261.Out;
  P7005.In_EquipEvents.6:= NOT P7005_VFD.IsFaulted;

// Function Call
P7005(
   In_p_EquipStatePB:= P7005_StatePB,
   In_P_ConvReqRun:= TRUE,
   In_ConvDwnStrmMtrStatus:= P7010_Status.Sts_IsRunning,
   In_ConvCrntExitPhotoEye:= PhotoEyes.PE_12301.Out, 
   In_SimActive:= System.Sys_SimActive,
   In_EquipInit:= GVL_IO.INIT,
   In_WakeSlpTrigArry:= P7005SleepWakeTrig,
   Cfg_EquipIndex := GVL_EquipArrays.nEquipIndex,
   Cfg_EquipLabel := cfgP7005Label,
   Cfg_EquipDefState:= System.ConvDefaultState,
   Cfg_EquipIntlksArry:= cfgP7005IntlksArry,
   Cfg_EquipEvntsArry:= cfgP7005EvntsArry,
   cfg_JamDetectTime:= cfgP7005JamDetectTime,
   Cfg_UseSleepTmr := TRUE,
   Cfg_UseStartUpDelay := TRUE,
   Cfg_StartUpDelayTime := T#500MS,
   Cfg_SleepWaitTime:= cfgP7005SleepTime,
   Sts_EquipState := P7005_Status);

//Motor Control
P7005_VFD(
   RunVelocity := DefaultVelocity,
   VelocityThreshold := DefaultVelocityThreshold,
   Reset := ResetAllDrives,
   RunRequest := (P7005.Out_ConvCrntMtr OR Test_VFD_P7005));
P7005_Status.Sts_IsRunning := P7005_VFD.IsRunning;
//----------------------------------------P7010--------------------------------------------------------------
P7010_StatePB.AutoPB := System.Cnvyr_Auto;
P7010_StatePB.ManPB := System.Cnvyr_Manual;
P7010_StatePB.ResetPB := System.Cnvyr_Reset;
P7010_StatePB.OfflinePB := System.Cnvyr_Offline;
P7010SleepWakeTrig[1] := PhotoEyes.PE_12301.Out_OffFltrd;
P7010SleepWakeTrig[2] := PhotoEyes.PE_12221.Out_OffFltrd;

// Initialize the Equipment Type
P7010_Status.Sts_EquipmentState.EquipType := E_EquipType.Conveyor;

// Interlocks
  P7010.In_EquipIntlks.2:= FALSE;
//Events
  P7010.In_EquipEvents.2:= GVL_IO.DS_P7010;
  P7010.In_EquipEvents.3:= System.SysEventsAllOk;
  P7010.In_EquipEvents.4:= NOT CommStatus.RIO12171_CommFault.Out;
  P7010.In_EquipEvents.5:= NOT GVL_IO.P7010_Faulted;

// Function Call
P7010(
   In_p_EquipStatePB:= P7010_StatePB,
   In_P_ConvReqRun:= TRUE,
   In_ConvDwnStrmMtrStatus:= P7015_Status.Sts_IsRunning,
   In_ConvCrntExitPhotoEye:= Photoeyes.PE_12231.Out,
   In_SimActive:= System.Sys_SimActive,
   In_EquipInit:= GVL_IO.INIT,
   In_WakeSlpTrigArry:= P7010SleepWakeTrig,
   Cfg_EquipIndex := GVL_EquipArrays.nEquipIndex,
   Cfg_EquipLabel := cfgP7010Label,
   Cfg_EquipDefState:= System.ConvDefaultState,
   Cfg_EquipIntlksArry:= cfgP7010IntlksArry,
   Cfg_EquipEvntsArry:= cfgP7010EvntsArry,
   cfg_JamDetectTime:= cfgP7010JamDetectTime,
   Cfg_UseSleepTmr := TRUE,
   Cfg_UseStartUpDelay := TRUE,
   Cfg_StartUpDelayTime := T#500MS,
   Cfg_SleepWaitTime:= cfgP7010SleepTime,
   Sts_EquipState := P7010_Status,
   Out_ConvCrntMtr => GVL_IO.P7010_RUN);

P7010_Status.Sts_IsRunning := GVL_IO.P7010_RUN;
//----------------------------------------P7015--------------------------------------------------------------
P7015_StatePB.AutoPB := System.Cnvyr_Auto;
P7015_StatePB.ManPB := System.Cnvyr_Manual;
P7015_StatePB.ResetPB := System.Cnvyr_Reset;
P7015_StatePB.OfflinePB := System.Cnvyr_Offline;
P7015SleepWakeTrig[1] := PhotoEyes.PE_12231.Out_OffFltrd;
P7015SleepWakeTrig[2] := PhotoEyes.PE_12301.Out_OffFltrd;

// Initialize the Equipment Type
P7015_Status.Sts_EquipmentState.EquipType := E_EquipType.Conveyor;

// Interlocks
  P7015.In_EquipIntlks.2:= FALSE;
//Events
  P7015.In_EquipEvents.2:= GVL_IO.DS_P7015;
  P7015.In_EquipEvents.3:= System.SysEventsAllOk;
  P7015.In_EquipEvents.4:= NOT CommStatus.RIO15181_CommFault.Out;
  P7015.In_EquipEvents.5:= NOT GVL_IO.P7015_Faulted;

// Function Call
P7015(
   In_p_EquipStatePB:= P7015_StatePB,
   In_P_ConvReqRun:= TRUE,
   In_ConvDwnStrmMtrStatus:= P7020_Status.Sts_IsRunning,
   In_ConvCrntExitPhotoEye:= Photoeyes.PE_15121.Out,
   In_SimActive:= System.Sys_SimActive,
   In_EquipInit:= GVL_IO.INIT,
   In_WakeSlpTrigArry:= P7015SleepWakeTrig,
   Cfg_EquipIndex := GVL_EquipArrays.nEquipIndex,
   Cfg_EquipLabel := cfgP7015Label,
   Cfg_EquipDefState:= System.ConvDefaultState,
   Cfg_EquipIntlksArry:= cfgP7015IntlksArry,
   Cfg_EquipEvntsArry:= cfgP7015EvntsArry,
   cfg_JamDetectTime:= cfgP7015JamDetectTime,
   Cfg_UseSleepTmr := TRUE,
   Cfg_UseStartUpDelay := TRUE,
   Cfg_StartUpDelayTime := T#500MS,
   Cfg_SleepWaitTime:= cfgP7015SleepTime,
   Sts_EquipState := P7015_Status,
   Out_ConvCrntMtr => GVL_IO.P7015_RUN);

P7015_Status.Sts_IsRunning := GVL_IO.P7015_RUN;
//----------------------------------------P7020--------------------------------------------------------------
P7020_StatePB.AutoPB := System.Cnvyr_Auto;
P7020_StatePB.ManPB := System.Cnvyr_Manual;
P7020_StatePB.ResetPB := System.Cnvyr_Reset;
P7020_StatePB.OfflinePB := System.Cnvyr_Offline;
P7020SleepWakeTrig[1] := PhotoEyes.PE_15121.Out_OffFltrd;
P7020SleepWakeTrig[2] := PhotoEyes.PE_12231.Out_OffFltrd;

// Initialize the Equipment Type
P7020_Status.Sts_EquipmentState.EquipType := E_EquipType.Conveyor;

// Interlocks
  P7020.In_EquipIntlks.2:= FALSE;
//Events
  P7020.In_EquipEvents.2:= GVL_IO.DS_P7020;
  P7020.In_EquipEvents.3:= System.SysEventsAllOk;
  P7020.In_EquipEvents.4:= NOT CommStatus.RIO15181_CommFault.Out;
  P7020.In_EquipEvents.5:= NOT GVL_IO.P7020_Faulted;
 

// Function Call
P7020(
   In_p_EquipStatePB:= P7020_StatePB,
   In_P_ConvReqRun:= TRUE,
   In_ConvDwnStrmMtrStatus:= P7025_Status.Sts_IsRunning,
   In_ConvCrntExitPhotoEye:= Photoeyes.PE_15181.Out,
   In_SimActive:= System.Sys_SimActive,
   In_EquipInit:= GVL_IO.INIT,
   In_WakeSlpTrigArry:= P7020SleepWakeTrig,
   Cfg_EquipIndex := GVL_EquipArrays.nEquipIndex,
   Cfg_EquipLabel := cfgP7020Label,
   Cfg_EquipDefState:= System.ConvDefaultState,
   Cfg_EquipIntlksArry:= cfgP7020IntlksArry,
   Cfg_EquipEvntsArry:= cfgP7020EvntsArry,
   cfg_JamDetectTime:= cfgP7020JamDetectTime,
   Cfg_UseSleepTmr := TRUE,
   Cfg_UseStartUpDelay := TRUE,
   Cfg_StartUpDelayTime := T#500MS,
   Cfg_SleepWaitTime:= cfgP7020SleepTime,
   Sts_EquipState := P7020_Status,
   Out_ConvCrntMtr => GVL_IO.P7020_RUN);

P7020_Status.Sts_IsRunning := GVL_IO.P7020_RUN;
//----------------------------------------P7025--------------------------------------------------------------
P7025_StatePB.AutoPB := System.Cnvyr_Auto;
P7025_StatePB.ManPB := System.Cnvyr_Manual;
P7025_StatePB.ResetPB := System.Cnvyr_Reset;
P7025_StatePB.OfflinePB := System.Cnvyr_Offline;
P7025SleepWakeTrig[1] := PhotoEyes.PE_15181.Out_OffFltrd;
P7025SleepWakeTrig[2] := PhotoEyes.PE_15121.Out_OffFltrd;

// Initialize the Equipment Type
P7025_Status.Sts_EquipmentState.EquipType := E_EquipType.Conveyor;

// Interlocks
  P7025.In_EquipIntlks.2:= FALSE;
//Events
  P7025.In_EquipEvents.2:=  GVL_IO.DS_P7025;
  P7025.In_EquipEvents.3:= System.SysEventsAllOk;
  P7025.In_EquipEvents.4:= NOT CommStatus.RIO15181_CommFault.Out;
  P7025.In_EquipEvents.5:= NOT GVL_IO.P7025_Faulted;

// Function Call
P7025(
   In_p_EquipStatePB:= P7025_StatePB,
   In_P_ConvReqRun:= TRUE,
   In_ConvDwnStrmMtrStatus:= P7030_Status.Sts_IsRunning,
   In_ConvCrntExitPhotoEye:= Photoeyes.PE_15261.Out,
   In_SimActive:= System.Sys_SimActive,
   In_EquipInit:= GVL_IO.INIT,
   In_WakeSlpTrigArry:= P7025SleepWakeTrig,
   Cfg_EquipIndex := GVL_EquipArrays.nEquipIndex,
   Cfg_EquipLabel := cfgP7025Label,
   Cfg_EquipDefState:= System.ConvDefaultState,
   Cfg_EquipIntlksArry:= cfgP7025IntlksArry,
   Cfg_EquipEvntsArry:= cfgP7025EvntsArry,
   cfg_JamDetectTime:= cfgP7025JamDetectTime,
   Cfg_UseSleepTmr := TRUE,
   Cfg_UseStartUpDelay := TRUE,
   Cfg_StartUpDelayTime := T#500MS,
   Cfg_SleepWaitTime:= cfgP7025SleepTime,
   Sts_EquipState := P7025_Status,
   Out_ConvCrntMtr => GVL_IO.P7025_RUN);

P7025_Status.Sts_IsRunning := GVL_IO.P7025_RUN;
//----------------------------------------P7030--------------------------------------------------------------
P7030_StatePB.AutoPB := System.Cnvyr_Auto;
P7030_StatePB.ManPB := System.Cnvyr_Manual;
P7030_StatePB.ResetPB := System.Cnvyr_Reset;
P7030_StatePB.OfflinePB := System.Cnvyr_Offline;
P7030SleepWakeTrig[1] := PhotoEyes.PE_15261.Out_OffFltrd;
P7030SleepWakeTrig[2] := PhotoEyes.PE_15181.Out_OffFltrd;
P7030SleepWakeTrig[3] := PhotoEyes.PE_16111.Out_OffFltrd;

// Initialize the Equipment Type
P7030_Status.Sts_EquipmentState.EquipType := E_EquipType.Conveyor;

// Interlocks
  P7030.In_EquipIntlks.2:= FALSE;
//Events
  P7030.In_EquipEvents.2:=  GVL_IO.DS_P7030;
  P7030.In_EquipEvents.3:= System.SysEventsAllOk;
  P7030.In_EquipEvents.4:= NOT CommStatus.RIO16171_CommFault.Out;
  P7030.In_EquipEvents.5:= NOT GVL_IO.P7030_Faulted;

// Function Call
P7030(
   In_p_EquipStatePB:= P7030_StatePB,
   In_P_ConvReqRun:= TRUE,
   In_ConvDwnStrmMtrStatus:= P7035_Status.Sts_IsRunning,
   In_ConvCrntExitPhotoEye:= Photoeyes.PE_16111.Out,
   In_SimActive:= System.Sys_SimActive,
   In_EquipInit:= GVL_IO.INIT,
   In_WakeSlpTrigArry:= P7030SleepWakeTrig,
   Cfg_EquipIndex := GVL_EquipArrays.nEquipIndex,
   Cfg_EquipLabel := cfgP7030Label,
   Cfg_EquipDefState:= System.ConvDefaultState,
   Cfg_EquipIntlksArry:= cfgP7030IntlksArry,
   Cfg_EquipEvntsArry:= cfgP7030EvntsArry,
   cfg_JamDetectTime:= cfgP7030JamDetectTime,
   Cfg_UseSleepTmr := TRUE,
   Cfg_UseStartUpDelay := TRUE,
   Cfg_StartUpDelayTime := T#500MS,
   Cfg_SleepWaitTime:= cfgP7030SleepTime,
   Sts_EquipState := P7030_Status,
   Out_ConvCrntMtr => GVL_IO.P7030_RUN);

P7030_Status.Sts_IsRunning := GVL_IO.P7030_RUN;
//----------------------------------------P7035--------------------------------------------------------------
P7035_StatePB.AutoPB := System.Cnvyr_Auto;
P7035_StatePB.ManPB := System.Cnvyr_Manual;
P7035_StatePB.ResetPB := System.Cnvyr_Reset;
P7035_StatePB.OfflinePB := System.Cnvyr_Offline;
P7035SleepWakeTrig[1] := PhotoEyes.PE_16111.Out_OffFltrd;
P7035SleepWakeTrig[2] := PhotoEyes.PE_15261.Out_OffFltrd;
P7035SleepWakeTrig[3] := PhotoEyes.PE_16301.Out_OffFltrd;

// Initialize the Equipment Type
P7035_Status.Sts_EquipmentState.EquipType := E_EquipType.Conveyor;

// Interlocks
  P7035.In_EquipIntlks.2:= FALSE;
  P7035.In_EquipIntlks.3:= ProxSensors.PX_16231_Extended.Out;
//Events
  P7035.In_EquipEvents.2:= GVL_IO.DS_P7035;
  P7035.In_EquipEvents.3:= System.SysEventsAllOk;
  P7035.In_EquipEvents.4:= NOT Photoeyes.PE_16181.Out; //Goes low when door drops
  P7035.In_EquipEvents.5:= NOT CommStatus.RIO16171_CommFault.Out;
  P7035.In_EquipEvents.6:= NOT GVL_IO.P7035_Faulted;

// Function Call
P7035(
   In_p_EquipStatePB:= P7035_StatePB,
   In_P_ConvReqRun:= TRUE,
   In_ConvDwnStrmMtrStatus:= P7040_VFD.IsRunning,
   In_ConvCrntExitPhotoEye:= Photoeyes.PE_16301.Out,
   In_SimActive:= System.Sys_SimActive,
   In_EquipInit:= GVL_IO.INIT,
   In_WakeSlpTrigArry:= P7035SleepWakeTrig,
   Cfg_EquipIndex := GVL_EquipArrays.nEquipIndex,
   Cfg_EquipLabel := cfgP7035Label,
   Cfg_EquipDefState:= System.ConvDefaultState,
   Cfg_EquipIntlksArry:= cfgP7035IntlksArry,
   Cfg_EquipEvntsArry:= cfgP7035EvntsArry,
   cfg_JamDetectTime:= cfgP7035JamDetectTime,
   Cfg_UseSleepTmr := TRUE,
   Cfg_UseStartUpDelay := TRUE,
   Cfg_StartUpDelayTime := T#500MS,
   Cfg_SleepWaitTime:= cfgP7035SleepTime,
   Sts_EquipState := P7035_Status,
   Out_ConvCrntMtr => GVL_IO.P7035_RUN);

P7035_Status.Sts_IsRunning := GVL_IO.P7035_RUN;
//----------------------------------------P7040--------------------------------------------------------------
P7040_StatePB.AutoPB := System.Cnvyr_Auto;
P7040_StatePB.ManPB := System.Cnvyr_Manual;
P7040_StatePB.ResetPB := System.Cnvyr_Reset;
P7040_StatePB.OfflinePB := System.Cnvyr_Offline;
P7040SleepWakeTrig[1] := PhotoEyes.PE_16301.Out_OffFltrd;
P7040SleepWakeTrig[2] := PhotoEyes.PE_16111.Out_OffFltrd;
P7040SleepWakeTrig[3] := PhotoEyes.PE_16131.Out_OffFltrd;

// Initialize the Equipment Type
P7040_Status.Sts_EquipmentState.EquipType := E_EquipType.Conveyor;

// Interlocks
  P7040.In_EquipIntlks.2:= FALSE;
//Events
  P7040.In_EquipEvents.2:=  GVL_IO.DS_P7040;
  P7040.In_EquipEvents.3:= System.SysEventsAllOk;
  P7040.In_EquipEvents.4:= NOT CommStatus.RIO16171_CommFault.Out;
  P7040.In_EquipEvents.5:= NOT P7040_VFD.IsFaulted;

// Function Call
P7040(
   In_p_EquipStatePB:= P7040_StatePB,
   In_P_ConvReqRun:= TRUE,
   In_ConvDwnStrmMtrStatus:= P7045_Status.Sts_IsRunning,
   In_ConvCrntExitPhotoEye:= Photoeyes.PE_16131.Out,
   In_SimActive:= System.Sys_SimActive,
   In_EquipInit:= GVL_IO.INIT,
   In_WakeSlpTrigArry:= P7040SleepWakeTrig,
   Cfg_EquipIndex := GVL_EquipArrays.nEquipIndex,
   Cfg_EquipLabel := cfgP7040Label,
   Cfg_EquipDefState:= System.ConvDefaultState,
   Cfg_EquipIntlksArry:= cfgP7040IntlksArry,
   Cfg_EquipEvntsArry:= cfgP7040EvntsArry,
   cfg_JamDetectTime:= cfgP7040JamDetectTime,
   Cfg_UseSleepTmr := TRUE,   
   Cfg_UseStartUpDelay := FALSE,
   Cfg_SleepWaitTime:= cfgP7040SleepTime,
   Sts_EquipState := P7040_Status);

//Motor Control
P7040_VFD(
   RunVelocity := DefaultVelocity,
   VelocityThreshold := DefaultVelocityThreshold,
   Reset := ResetAllDrives,
   RunRequest := (P7040.Out_ConvCrntMtr OR Test_VFD_P7040));
P7040_Status.Sts_IsRunning := P7040_VFD.IsRunning;

//----------------------------------------P7045--------------------------------------------------------------
P7045_StatePB.AutoPB := System.Cnvyr_Auto;
P7045_StatePB.ManPB := System.Cnvyr_Manual;
P7045_StatePB.ResetPB := System.Cnvyr_Reset;
P7045_StatePB.OfflinePB := System.Cnvyr_Offline;
P7045SleepWakeTrig[1] := PhotoEyes.PE_16131.Out_OffFltrd;
P7045SleepWakeTrig[2] := PhotoEyes.PE_16301.Out_OffFltrd;

GVL_IO.To205_P7045_SendingProduct:= P7045_Status.Sts_IsRunning OR P7040_Status.Sts_IsRunning OR P7035_Status.Sts_IsRunning OR PhotoEyes.PE_16301.Out OR PhotoEyes.PE_16131.Out_OffFltrd;;

// Initialize the Equipment Type
P7045_Status.Sts_EquipmentState.EquipType := E_EquipType.Conveyor;

// Interlocks
  P7045.In_EquipIntlks.2:= FALSE;
//Events
  P7045.In_EquipEvents.2:=  GVL_IO.DS_P7045;
  P7045.In_EquipEvents.3:= System.SysEventsAllOk;
  P7045.In_EquipEvents.4:= ProxSensors.PX_16231_Extended.Out;
  P7045.In_EquipEvents.5:= NOT CommStatus.RIO16171_CommFault.Out;
  P7045.In_EquipEvents.6:= NOT GVL_IO.P7030_Faulted;

// Function Call
P7045(
   In_p_EquipStatePB:= P7045_StatePB,
   In_P_ConvReqRun:= TRUE,
   In_ConvDwnStrmMtrStatus:= GVL_IO.From205_P2012_IsRunning,
   In_ConvCrntExitPhotoEye:= Photoeyes.PE_16201.Out,
   In_SimActive:= System.Sys_SimActive,
   In_EquipInit:= GVL_IO.INIT,
   In_WakeSlpTrigArry:= P7045SleepWakeTrig,
   Cfg_EquipIndex := GVL_EquipArrays.nEquipIndex,
   Cfg_EquipLabel := cfgP7045Label,
   Cfg_EquipDefState:= System.ConvDefaultState,
   Cfg_EquipIntlksArry:= cfgP7045IntlksArry,
   Cfg_EquipEvntsArry:= cfgP7045EvntsArry,
   cfg_JamDetectTime:= cfgP7045JamDetectTime,
   Cfg_UseSleepTmr := TRUE,
   Cfg_SleepWaitTime:= cfgP7045SleepTime,
   Sts_EquipState := P7045_Status,
   Out_ConvCrntMtr => GVL_IO.P7045_RUN);

P7045_Status.Sts_IsRunning := GVL_IO.P7045_RUN;


	
//Equipment arrays
//Conveyors Incoming 6000 (Blue line)
//Transport
//P6005
//    Remote Index Check
IF Conveyors.P6005_Status.Sts_EquipmentState.Index > 0 THEN
  IF GVL_EquipArrays.aEquipStatusArray_Out[Conveyors.P6005_Status.Sts_EquipmentState.Index].RemIndex <> 0 THEN
      IF Conveyors.P6005_Status.Sts_EquipmentState.RemIndex = 0 THEN
          Conveyors.P6005_Status.Sts_EquipmentState.RemIndex := GVL_EquipArrays.aEquipStatusArray_Out[Conveyors.P6005_Status.Sts_EquipmentState.Index].RemIndex;
      END_IF
  END_IF
  //    Last Operational State Check
  IF GVL_EquipArrays.aEquipStatusArray_Out[Conveyors.P6005_Status.Sts_EquipmentState.Index].LstOperState <> Conveyors.P6005_Status.Sts_EquipmentState.LstOperState THEN
      Conveyors.P6005_Status.Sts_EquipmentState.LstOperState := GVL_EquipArrays.aEquipStatusArray_In[Conveyors.P6005_Status.Sts_EquipmentState.Index].LstOperState;
  END_IF
  //Prepare the Equipment Status data item
  GVL_EquipArrays.aEquipStatusArray_In[Conveyors.P6005_Status.Sts_EquipmentState.Index] := Conveyors.P6005_Status.Sts_EquipmentState;
END_IF

//Spiral
//P6010
//    Remote Index Check
IF Conveyors.P6010_Status.Sts_EquipmentState.Index > 0 THEN
  IF GVL_EquipArrays.aEquipStatusArray_Out[Conveyors.P6010_Status.Sts_EquipmentState.Index].RemIndex <> 0 THEN
      IF Conveyors.P6010_Status.Sts_EquipmentState.RemIndex = 0 THEN
          Conveyors.P6010_Status.Sts_EquipmentState.RemIndex := GVL_EquipArrays.aEquipStatusArray_Out[Conveyors.P6010_Status.Sts_EquipmentState.Index].RemIndex;
      END_IF
  END_IF
  //    Last Operational State Check
  IF GVL_EquipArrays.aEquipStatusArray_Out[Conveyors.P6010_Status.Sts_EquipmentState.Index].LstOperState <> Conveyors.P6010_Status.Sts_EquipmentState.LstOperState THEN
      Conveyors.P6010_Status.Sts_EquipmentState.LstOperState := GVL_EquipArrays.aEquipStatusArray_In[Conveyors.P6010_Status.Sts_EquipmentState.Index].LstOperState;
  END_IF
  //Prepare the Equipment Status data item
  GVL_EquipArrays.aEquipStatusArray_In[Conveyors.P6010_Status.Sts_EquipmentState.Index] := Conveyors.P6010_Status.Sts_EquipmentState;
END_IF



//Transport
//P6015
//    Remote Index Check
IF Conveyors.P6015_Status.Sts_EquipmentState.Index > 0 THEN
  IF GVL_EquipArrays.aEquipStatusArray_Out[Conveyors.P6015_Status.Sts_EquipmentState.Index].RemIndex <> 0 THEN
      IF Conveyors.P6015_Status.Sts_EquipmentState.RemIndex = 0 THEN
          Conveyors.P6015_Status.Sts_EquipmentState.RemIndex := GVL_EquipArrays.aEquipStatusArray_Out[Conveyors.P6015_Status.Sts_EquipmentState.Index].RemIndex;
      END_IF
  END_IF
  //    Last Operational State Check
  IF GVL_EquipArrays.aEquipStatusArray_Out[Conveyors.P6015_Status.Sts_EquipmentState.Index].LstOperState <> Conveyors.P6015_Status.Sts_EquipmentState.LstOperState THEN
      Conveyors.P6015_Status.Sts_EquipmentState.LstOperState := GVL_EquipArrays.aEquipStatusArray_In[Conveyors.P6015_Status.Sts_EquipmentState.Index].LstOperState;
  END_IF
  //Prepare the Equipment Status data item
  GVL_EquipArrays.aEquipStatusArray_In[Conveyors.P6015_Status.Sts_EquipmentState.Index] := Conveyors.P6015_Status.Sts_EquipmentState;
END_IF

//P6020
//    Remote Index Check
IF Conveyors.P6020_Status.Sts_EquipmentState.Index > 0 THEN
  IF GVL_EquipArrays.aEquipStatusArray_Out[Conveyors.P6020_Status.Sts_EquipmentState.Index].RemIndex <> 0 THEN
      IF Conveyors.P6020_Status.Sts_EquipmentState.RemIndex = 0 THEN
          Conveyors.P6020_Status.Sts_EquipmentState.RemIndex := GVL_EquipArrays.aEquipStatusArray_Out[Conveyors.P6020_Status.Sts_EquipmentState.Index].RemIndex;
      END_IF
  END_IF
  //    Last Operational State Check
  IF GVL_EquipArrays.aEquipStatusArray_Out[Conveyors.P6020_Status.Sts_EquipmentState.Index].LstOperState <> Conveyors.P6020_Status.Sts_EquipmentState.LstOperState THEN
      Conveyors.P6020_Status.Sts_EquipmentState.LstOperState := GVL_EquipArrays.aEquipStatusArray_In[Conveyors.P6020_Status.Sts_EquipmentState.Index].LstOperState;
  END_IF
  //Prepare the Equipment Status data item
  GVL_EquipArrays.aEquipStatusArray_In[Conveyors.P6020_Status.Sts_EquipmentState.Index] := Conveyors.P6020_Status.Sts_EquipmentState;
END_IF

//P6025
//    Remote Index Check
IF Conveyors.P6025_Status.Sts_EquipmentState.Index > 0 THEN
  IF GVL_EquipArrays.aEquipStatusArray_Out[Conveyors.P6025_Status.Sts_EquipmentState.Index].RemIndex <> 0 THEN
      IF Conveyors.P6025_Status.Sts_EquipmentState.RemIndex = 0 THEN
          Conveyors.P6025_Status.Sts_EquipmentState.RemIndex := GVL_EquipArrays.aEquipStatusArray_Out[Conveyors.P6025_Status.Sts_EquipmentState.Index].RemIndex;
      END_IF
  END_IF
  //    Last Operational State Check
  IF GVL_EquipArrays.aEquipStatusArray_Out[Conveyors.P6025_Status.Sts_EquipmentState.Index].LstOperState <> Conveyors.P6025_Status.Sts_EquipmentState.LstOperState THEN
      Conveyors.P6025_Status.Sts_EquipmentState.LstOperState := GVL_EquipArrays.aEquipStatusArray_In[Conveyors.P6025_Status.Sts_EquipmentState.Index].LstOperState;
  END_IF
  //Prepare the Equipment Status data item
  GVL_EquipArrays.aEquipStatusArray_In[Conveyors.P6025_Status.Sts_EquipmentState.Index] := Conveyors.P6025_Status.Sts_EquipmentState;
END_IF

//P6030
//    Remote Index Check
IF Conveyors.P6030_Status.Sts_EquipmentState.Index > 0 THEN
  IF GVL_EquipArrays.aEquipStatusArray_Out[Conveyors.P6030_Status.Sts_EquipmentState.Index].RemIndex <> 0 THEN
      IF Conveyors.P6030_Status.Sts_EquipmentState.RemIndex = 0 THEN
          Conveyors.P6030_Status.Sts_EquipmentState.RemIndex := GVL_EquipArrays.aEquipStatusArray_Out[Conveyors.P6030_Status.Sts_EquipmentState.Index].RemIndex;
      END_IF
  END_IF
  //    Last Operational State Check
  IF GVL_EquipArrays.aEquipStatusArray_Out[Conveyors.P6030_Status.Sts_EquipmentState.Index].LstOperState <> Conveyors.P6030_Status.Sts_EquipmentState.LstOperState THEN
      Conveyors.P6030_Status.Sts_EquipmentState.LstOperState := GVL_EquipArrays.aEquipStatusArray_In[Conveyors.P6030_Status.Sts_EquipmentState.Index].LstOperState;
  END_IF
  //Prepare the Equipment Status data item
  GVL_EquipArrays.aEquipStatusArray_In[Conveyors.P6030_Status.Sts_EquipmentState.Index] := Conveyors.P6030_Status.Sts_EquipmentState;
END_IF

//P6035
//    Remote Index Check
IF Conveyors.P6035_Status.Sts_EquipmentState.Index > 0 THEN
  IF GVL_EquipArrays.aEquipStatusArray_Out[Conveyors.P6035_Status.Sts_EquipmentState.Index].RemIndex <> 0 THEN
      IF Conveyors.P6035_Status.Sts_EquipmentState.RemIndex = 0 THEN
          Conveyors.P6035_Status.Sts_EquipmentState.RemIndex := GVL_EquipArrays.aEquipStatusArray_Out[Conveyors.P6035_Status.Sts_EquipmentState.Index].RemIndex;
      END_IF
  END_IF
  //    Last Operational State Check
  IF GVL_EquipArrays.aEquipStatusArray_Out[Conveyors.P6035_Status.Sts_EquipmentState.Index].LstOperState <> Conveyors.P6035_Status.Sts_EquipmentState.LstOperState THEN
      Conveyors.P6035_Status.Sts_EquipmentState.LstOperState := GVL_EquipArrays.aEquipStatusArray_In[Conveyors.P6035_Status.Sts_EquipmentState.Index].LstOperState;
  END_IF
  //Prepare the Equipment Status data item
  GVL_EquipArrays.aEquipStatusArray_In[Conveyors.P6035_Status.Sts_EquipmentState.Index] := Conveyors.P6035_Status.Sts_EquipmentState;
END_IF

//Spiral
//P6045
//    Remote Index Check
IF Conveyors.P6045_Status.Sts_EquipmentState.Index > 0 THEN
  IF GVL_EquipArrays.aEquipStatusArray_Out[Conveyors.P6045_Status.Sts_EquipmentState.Index].RemIndex <> 0 THEN
      IF Conveyors.P6045_Status.Sts_EquipmentState.RemIndex = 0 THEN
          Conveyors.P6045_Status.Sts_EquipmentState.RemIndex := GVL_EquipArrays.aEquipStatusArray_Out[Conveyors.P6045_Status.Sts_EquipmentState.Index].RemIndex;
      END_IF
  END_IF
  //    Last Operational State Check
  IF GVL_EquipArrays.aEquipStatusArray_Out[Conveyors.P6045_Status.Sts_EquipmentState.Index].LstOperState <> Conveyors.P6045_Status.Sts_EquipmentState.LstOperState THEN
      Conveyors.P6045_Status.Sts_EquipmentState.LstOperState := GVL_EquipArrays.aEquipStatusArray_In[Conveyors.P6045_Status.Sts_EquipmentState.Index].LstOperState;
  END_IF
  //Prepare the Equipment Status data item
  GVL_EquipArrays.aEquipStatusArray_In[Conveyors.P6045_Status.Sts_EquipmentState.Index] := Conveyors.P6045_Status.Sts_EquipmentState;
END_IF

//Sorter
//P6040
//    Remote Index Check
IF Conveyors.P6040_Status.Sts_EquipmentState.Index > 0 THEN
  IF GVL_EquipArrays.aEquipStatusArray_Out[Conveyors.P6040_Status.Sts_EquipmentState.Index].RemIndex <> 0 THEN
      IF Conveyors.P6040_Status.Sts_EquipmentState.RemIndex = 0 THEN
          Conveyors.P6040_Status.Sts_EquipmentState.RemIndex := GVL_EquipArrays.aEquipStatusArray_Out[Conveyors.P6040_Status.Sts_EquipmentState.Index].RemIndex;
      END_IF
  END_IF
  //    Last Operational State Check
  IF GVL_EquipArrays.aEquipStatusArray_Out[Conveyors.P6040_Status.Sts_EquipmentState.Index].LstOperState <> Conveyors.P6040_Status.Sts_EquipmentState.LstOperState THEN
      Conveyors.P6040_Status.Sts_EquipmentState.LstOperState := GVL_EquipArrays.aEquipStatusArray_In[Conveyors.P6040_Status.Sts_EquipmentState.Index].LstOperState;
  END_IF
  //Prepare the Equipment Status data item
  GVL_EquipArrays.aEquipStatusArray_In[Conveyors.P6040_Status.Sts_EquipmentState.Index] := Conveyors.P6040_Status.Sts_EquipmentState;
END_IF

//Conveyors Outgoing 7000 (Orange line)
//Loading Zone
//P7004
//    Remote Index Check
IF Conveyors.P7004_Status.Sts_EquipmentState.Index > 0 THEN
  IF GVL_EquipArrays.aEquipStatusArray_Out[Conveyors.P7004_Status.Sts_EquipmentState.Index].RemIndex <> 0 THEN
      IF Conveyors.P7004_Status.Sts_EquipmentState.RemIndex = 0 THEN
          Conveyors.P7004_Status.Sts_EquipmentState.RemIndex := GVL_EquipArrays.aEquipStatusArray_Out[Conveyors.P7004_Status.Sts_EquipmentState.Index].RemIndex;
      END_IF
  END_IF
  //    Last Operational State Check
  IF GVL_EquipArrays.aEquipStatusArray_Out[Conveyors.P7004_Status.Sts_EquipmentState.Index].LstOperState <> Conveyors.P7004_Status.Sts_EquipmentState.LstOperState THEN
      Conveyors.P7004_Status.Sts_EquipmentState.LstOperState := GVL_EquipArrays.aEquipStatusArray_In[Conveyors.P7004_Status.Sts_EquipmentState.Index].LstOperState;
  END_IF
  //Prepare the Equipment Status data item
  GVL_EquipArrays.aEquipStatusArray_In[Conveyors.P7004_Status.Sts_EquipmentState.Index] := Conveyors.P7004_Status.Sts_EquipmentState;
     // Overwriter Conv label with EquipID
  GVL_EquipArrays.aEquipStatusArray_In[Conveyors.P7004_Status.Sts_EquipmentState.Index].Label := '00063';
END_IF

//Spiral
//P7005
//    Remote Index Check
IF Conveyors.P7005_Status.Sts_EquipmentState.Index > 0 THEN
  IF GVL_EquipArrays.aEquipStatusArray_Out[Conveyors.P7005_Status.Sts_EquipmentState.Index].RemIndex <> 0 THEN
      IF Conveyors.P7005_Status.Sts_EquipmentState.RemIndex = 0 THEN
          Conveyors.P7005_Status.Sts_EquipmentState.RemIndex := GVL_EquipArrays.aEquipStatusArray_Out[Conveyors.P7005_Status.Sts_EquipmentState.Index].RemIndex;
      END_IF
  END_IF
  //    Last Operational State Check
  IF GVL_EquipArrays.aEquipStatusArray_Out[Conveyors.P7005_Status.Sts_EquipmentState.Index].LstOperState <> Conveyors.P7005_Status.Sts_EquipmentState.LstOperState THEN
      Conveyors.P7005_Status.Sts_EquipmentState.LstOperState := GVL_EquipArrays.aEquipStatusArray_In[Conveyors.P7005_Status.Sts_EquipmentState.Index].LstOperState;
  END_IF
  //Prepare the Equipment Status data item
  GVL_EquipArrays.aEquipStatusArray_In[Conveyors.P7005_Status.Sts_EquipmentState.Index] := Conveyors.P7005_Status.Sts_EquipmentState;
END_IF

//Transport
//P7010
//    Remote Index Check
IF Conveyors.P7010_Status.Sts_EquipmentState.Index > 0 THEN
  IF GVL_EquipArrays.aEquipStatusArray_Out[Conveyors.P7010_Status.Sts_EquipmentState.Index].RemIndex <> 0 THEN
      IF Conveyors.P7010_Status.Sts_EquipmentState.RemIndex = 0 THEN
          Conveyors.P7010_Status.Sts_EquipmentState.RemIndex := GVL_EquipArrays.aEquipStatusArray_Out[Conveyors.P7010_Status.Sts_EquipmentState.Index].RemIndex;
      END_IF
  END_IF
  //    Last Operational State Check
  IF GVL_EquipArrays.aEquipStatusArray_Out[Conveyors.P7010_Status.Sts_EquipmentState.Index].LstOperState <> Conveyors.P7010_Status.Sts_EquipmentState.LstOperState THEN
      Conveyors.P7010_Status.Sts_EquipmentState.LstOperState := GVL_EquipArrays.aEquipStatusArray_In[Conveyors.P7010_Status.Sts_EquipmentState.Index].LstOperState;
  END_IF
  //Prepare the Equipment Status data item
  GVL_EquipArrays.aEquipStatusArray_In[Conveyors.P7010_Status.Sts_EquipmentState.Index] := Conveyors.P7010_Status.Sts_EquipmentState;
END_IF

//P7015
//    Remote Index Check
IF Conveyors.P7015_Status.Sts_EquipmentState.Index > 0 THEN
  IF GVL_EquipArrays.aEquipStatusArray_Out[Conveyors.P7015_Status.Sts_EquipmentState.Index].RemIndex <> 0 THEN
      IF Conveyors.P7015_Status.Sts_EquipmentState.RemIndex = 0 THEN
          Conveyors.P7015_Status.Sts_EquipmentState.RemIndex := GVL_EquipArrays.aEquipStatusArray_Out[Conveyors.P7015_Status.Sts_EquipmentState.Index].RemIndex;
      END_IF
  END_IF
  //    Last Operational State Check
  IF GVL_EquipArrays.aEquipStatusArray_Out[Conveyors.P7015_Status.Sts_EquipmentState.Index].LstOperState <> Conveyors.P7015_Status.Sts_EquipmentState.LstOperState THEN
      Conveyors.P7015_Status.Sts_EquipmentState.LstOperState := GVL_EquipArrays.aEquipStatusArray_In[Conveyors.P7015_Status.Sts_EquipmentState.Index].LstOperState;
  END_IF
  //Prepare the Equipment Status data item
  GVL_EquipArrays.aEquipStatusArray_In[Conveyors.P7015_Status.Sts_EquipmentState.Index] := Conveyors.P7015_Status.Sts_EquipmentState;
END_IF

//P7020
//    Remote Index Check
IF Conveyors.P7020_Status.Sts_EquipmentState.Index > 0 THEN
  IF GVL_EquipArrays.aEquipStatusArray_Out[Conveyors.P7020_Status.Sts_EquipmentState.Index].RemIndex <> 0 THEN
      IF Conveyors.P7020_Status.Sts_EquipmentState.RemIndex = 0 THEN
          Conveyors.P7020_Status.Sts_EquipmentState.RemIndex := GVL_EquipArrays.aEquipStatusArray_Out[Conveyors.P7020_Status.Sts_EquipmentState.Index].RemIndex;
      END_IF
  END_IF
  //    Last Operational State Check
  IF GVL_EquipArrays.aEquipStatusArray_Out[Conveyors.P7020_Status.Sts_EquipmentState.Index].LstOperState <> Conveyors.P7020_Status.Sts_EquipmentState.LstOperState THEN
      Conveyors.P7020_Status.Sts_EquipmentState.LstOperState := GVL_EquipArrays.aEquipStatusArray_In[Conveyors.P7020_Status.Sts_EquipmentState.Index].LstOperState;
  END_IF
  //Prepare the Equipment Status data item
  GVL_EquipArrays.aEquipStatusArray_In[Conveyors.P7020_Status.Sts_EquipmentState.Index] := Conveyors.P7020_Status.Sts_EquipmentState;
END_IF

//P7025
//    Remote Index Check
IF Conveyors.P7025_Status.Sts_EquipmentState.Index > 0 THEN
  IF GVL_EquipArrays.aEquipStatusArray_Out[Conveyors.P7025_Status.Sts_EquipmentState.Index].RemIndex <> 0 THEN
      IF Conveyors.P7025_Status.Sts_EquipmentState.RemIndex = 0 THEN
          Conveyors.P7025_Status.Sts_EquipmentState.RemIndex := GVL_EquipArrays.aEquipStatusArray_Out[Conveyors.P7025_Status.Sts_EquipmentState.Index].RemIndex;
      END_IF
  END_IF
  //    Last Operational State Check
  IF GVL_EquipArrays.aEquipStatusArray_Out[Conveyors.P7025_Status.Sts_EquipmentState.Index].LstOperState <> Conveyors.P7025_Status.Sts_EquipmentState.LstOperState THEN
      Conveyors.P7025_Status.Sts_EquipmentState.LstOperState := GVL_EquipArrays.aEquipStatusArray_In[Conveyors.P7025_Status.Sts_EquipmentState.Index].LstOperState;
  END_IF
  //Prepare the Equipment Status data item
  GVL_EquipArrays.aEquipStatusArray_In[Conveyors.P7025_Status.Sts_EquipmentState.Index] := Conveyors.P7025_Status.Sts_EquipmentState;
END_IF

//P7030
//    Remote Index Check
IF Conveyors.P7030_Status.Sts_EquipmentState.Index > 0 THEN
  IF GVL_EquipArrays.aEquipStatusArray_Out[Conveyors.P7030_Status.Sts_EquipmentState.Index].RemIndex <> 0 THEN
      IF Conveyors.P7030_Status.Sts_EquipmentState.RemIndex = 0 THEN
          Conveyors.P7030_Status.Sts_EquipmentState.RemIndex := GVL_EquipArrays.aEquipStatusArray_Out[Conveyors.P7030_Status.Sts_EquipmentState.Index].RemIndex;
      END_IF
  END_IF
  //    Last Operational State Check
  IF GVL_EquipArrays.aEquipStatusArray_Out[Conveyors.P7030_Status.Sts_EquipmentState.Index].LstOperState <> Conveyors.P7030_Status.Sts_EquipmentState.LstOperState THEN
      Conveyors.P7030_Status.Sts_EquipmentState.LstOperState := GVL_EquipArrays.aEquipStatusArray_In[Conveyors.P7030_Status.Sts_EquipmentState.Index].LstOperState;
  END_IF
  //Prepare the Equipment Status data item
  GVL_EquipArrays.aEquipStatusArray_In[Conveyors.P7030_Status.Sts_EquipmentState.Index] := Conveyors.P7030_Status.Sts_EquipmentState;
END_IF

//P7035
//    Remote Index Check
IF Conveyors.P7035_Status.Sts_EquipmentState.Index > 0 THEN
  IF GVL_EquipArrays.aEquipStatusArray_Out[Conveyors.P7035_Status.Sts_EquipmentState.Index].RemIndex <> 0 THEN
      IF Conveyors.P7035_Status.Sts_EquipmentState.RemIndex = 0 THEN
          Conveyors.P7035_Status.Sts_EquipmentState.RemIndex := GVL_EquipArrays.aEquipStatusArray_Out[Conveyors.P7035_Status.Sts_EquipmentState.Index].RemIndex;
      END_IF
  END_IF
  //    Last Operational State Check
  IF GVL_EquipArrays.aEquipStatusArray_Out[Conveyors.P7035_Status.Sts_EquipmentState.Index].LstOperState <> Conveyors.P7035_Status.Sts_EquipmentState.LstOperState THEN
      Conveyors.P7035_Status.Sts_EquipmentState.LstOperState := GVL_EquipArrays.aEquipStatusArray_In[Conveyors.P7035_Status.Sts_EquipmentState.Index].LstOperState;
  END_IF
  //Prepare the Equipment Status data item
  GVL_EquipArrays.aEquipStatusArray_In[Conveyors.P7035_Status.Sts_EquipmentState.Index] := Conveyors.P7035_Status.Sts_EquipmentState;
END_IF

//Spiral
//P7040
//    Remote Index Check
IF Conveyors.P7040_Status.Sts_EquipmentState.Index > 0 THEN
  IF GVL_EquipArrays.aEquipStatusArray_Out[Conveyors.P7040_Status.Sts_EquipmentState.Index].RemIndex <> 0 THEN
      IF Conveyors.P7040_Status.Sts_EquipmentState.RemIndex = 0 THEN
          Conveyors.P7040_Status.Sts_EquipmentState.RemIndex := GVL_EquipArrays.aEquipStatusArray_Out[Conveyors.P7040_Status.Sts_EquipmentState.Index].RemIndex;
      END_IF
  END_IF
  //    Last Operational State Check
  IF GVL_EquipArrays.aEquipStatusArray_Out[Conveyors.P7040_Status.Sts_EquipmentState.Index].LstOperState <> Conveyors.P7040_Status.Sts_EquipmentState.LstOperState THEN
      Conveyors.P7040_Status.Sts_EquipmentState.LstOperState := GVL_EquipArrays.aEquipStatusArray_In[Conveyors.P7040_Status.Sts_EquipmentState.Index].LstOperState;
  END_IF
  //Prepare the Equipment Status data item
  GVL_EquipArrays.aEquipStatusArray_In[Conveyors.P7040_Status.Sts_EquipmentState.Index] := Conveyors.P7040_Status.Sts_EquipmentState;
END_IF



//Transport
//P7045
//    Remote Index Check
IF Conveyors.P7045_Status.Sts_EquipmentState.Index > 0 THEN
  IF GVL_EquipArrays.aEquipStatusArray_Out[Conveyors.P7045_Status.Sts_EquipmentState.Index].RemIndex <> 0 THEN
      IF Conveyors.P7045_Status.Sts_EquipmentState.RemIndex = 0 THEN
          Conveyors.P7045_Status.Sts_EquipmentState.RemIndex := GVL_EquipArrays.aEquipStatusArray_Out[Conveyors.P7045_Status.Sts_EquipmentState.Index].RemIndex;
      END_IF
  END_IF
  //    Last Operational State Check
  IF GVL_EquipArrays.aEquipStatusArray_Out[Conveyors.P7045_Status.Sts_EquipmentState.Index].LstOperState <> Conveyors.P7045_Status.Sts_EquipmentState.LstOperState THEN
      Conveyors.P7045_Status.Sts_EquipmentState.LstOperState := GVL_EquipArrays.aEquipStatusArray_In[Conveyors.P7045_Status.Sts_EquipmentState.Index].LstOperState;
  END_IF
  //Prepare the Equipment Status data item
  GVL_EquipArrays.aEquipStatusArray_In[Conveyors.P7045_Status.Sts_EquipmentState.Index] := Conveyors.P7045_Status.Sts_EquipmentState;
END_IF

END_PROGRAM

// ---- POUs/FunctionBlocks/Conveyance/FB_CnvyrCnfig_1.TcPOU
FUNCTION_BLOCK FB_CnvyrCnfig_1

(* Standard Conveyor Set up,
	Uses Interlocks. Has 14 that can be assigned that are conveyor specific and a common interlock for exit conveyor PE and Dwn Stream MTR status
	Has an interlock for System.SysIntlksAllOk
	Doesn't use Start Conditions  
	Uses Events and has 15 that can be assigned that are conveyor specific and a common event for the exit conveyor PE Jam detected fault  *)
(* End Conveyor Set up,
	This configuration doesn't use the downstream motor status
	Uses Interlocks. Has 14 that can be assigned that are conveyor specific and a common interlock for conveyor full using the exit PE of this conveyor
	Has an interlock for System.SysIntlksAllOk
	Doesn't use Start Conditions  
	Uses Events and has 16 that can be assigned that are conveyor specific *)
(* Slave Conveyor Set up,
	Uses Interlocks. Has 14 that can be assigned that are conveyor specific and a common interlock for Dwn Stream MTR status
	Has an interlock for System.SysIntlksAllOk
	Doesn't use Start Conditions  
	Uses Events and has 16 that can be assigned that are conveyor specifi  *)

VAR_IN_OUT
	CFG_EquipIndex				: DINT;	// Index used for local Equipment status array
	{attribute 'OPC.UA.DA' := '1'}
	Sts_EquipState				: ST_EquipmentStatus;		// State Status
END_VAR
VAR_INPUT
	{attribute 'OPC.UA.DA' := '1'}
	In_o_EquipStatePB			: ST_StateCntrlPB;		// Hmi push butons to change states
	In_p_EquipStatePB			: ST_StateCntrlPB;		// programming to change states
	In_P_ConvReqRun				: BOOL;		// Input to start output if in auto and conditions are met
	In_ConvDwnStrmMtrStatus		: BOOL;		// The Down Stearm Motors Status (0= OFF, 1= ON/Running)
	In_ConvCrntExitPhotoEye		: BOOL;		// The Current Photo Eye (1= blocked)
	In_SimActive				: BOOL;
	In_EquipInit					: BOOL;		// Initialise;
	In_EquipMtrFdbck			: BOOL := FALSE;	// Motor Running Feedback (1 = Running), VFD or Contactor
	Cfg_EquipDefState			: E_StateCntrl;
	{attribute 'OPC.UA.DA' := '1'}
	Cfg_EquipLabel				: STRING(20);		// Label of the conveyor
	Cfg_UseMtrFdbck				: BOOL := FALSE;	// Use Feedback from Contactor or VFD 
	Cfg_UseStartUpDelay			: BOOL := FALSE;	// Use a Start-up Delay
	Cfg_StartUpDelayTime		: TIME := T#1S;		// Start-up delay time
	Cfg_InvertMotorOut          : BOOL := FALSE;
	Cfg_ConvType				: E_ConvType := E_ConvType.standard;	// Default to a standard conveyor type
	Cfg_JamDetectTime			: TIME;
	
	// Events
	In_EquipEvents				: UINT;		// Events that are specific to the instance of the conveyor
	{attribute 'OPC.UA.DA' := '0'}
	Cfg_EquipEvntsArry			: ARRAY [0..15] OF ST_CfgEvents;
	
	// Interlocks that can be Instance Specific
	In_EquipIntlks				: UINT;		// Interlock that is specific to the instance of the conveyor
	{attribute 'OPC.UA.DA' := '0'}
	Cfg_EquipIntlksArry			: ARRAY [0..15] OF ST_CfgEvents;		// Descriptions of the Interlock 
	
	// Sleep Timer	
	Cfg_UseSleepTmr				: BOOL;	// Configure sleep or not sleep this conveyor
	In_WakeSlpTrigArry			: ARRAY [1..5] OF BOOL;		// Input to watch (or wake) for sleep timer
	Cfg_SleepWaitTime			: TIME;		// Time to Wait after last Input before sleeping
	
END_VAR
VAR_OUTPUT
	{attribute 'OPC.UA.DA' := '1'}
	Out_ConvCrntMtr				: BOOL;		// Run command for the current motor
	{attribute 'OPC.UA.DA' := '1'}
	Out_ConvCrntMtr_Raw			: BOOL;		// Run command for the current motor
	{attribute 'OPC.UA.DA' := '1'}
	Sts_ConvCrntMtr				: BOOL;		// Status showing that current motor is running
	{attribute 'OPC.UA.DA' := '1'}
	Sts_ConvSleepingActive		: BOOL;
	{attribute 'OPC.UA.DA' := '1'}
	Sts_All_Intlks_OK			: BOOL;		// Status bit to show that all interloks are good to Run 
	{attribute 'OPC.UA.DA' := '1'}
	Sts_FaultActive				: BOOL;	// Status Bit Showing that a fault is present (0= No Active Faults, 1= Fault Active)
	{attribute 'OPC.UA.DA' := '1'}
	Sts_WarnActive				: BOOL;	// Status Bit Showing that a warning is present (0= No Active Warnings, 1= Warning Active)
	{attribute 'OPC.UA.DA' := '1'}
	Sts_All_Evnts_OK			: BOOL;		// Status Bit Showing that ALL Events are OK to RUN (0= Event Present, 1= OK to Run)
	{attribute 'OPC.UA.DA' := '1'}
	Sts_IntlksArry				: ARRAY[0..15] OF ST_EventSts;		// Interlock status 0 to 15 Input
	{attribute 'OPC.UA.DA' := '1'}
	Sts_FaultsArry				: ARRAY[0..15] OF ST_EventSts;	// Status of each Fault Event State (0= OFF, 1=ON)
	{attribute 'OPC.UA.DA' := '1'}
	Sts_WarnsArry				: ARRAY[0..15] OF ST_EventSts;		// Status of each Warning Event State (0= OFF, 1=ON)
	{attribute 'OPC.UA.DA' := '0'}
	Sts_EvntsArry				: ARRAY[0..15] OF ST_EventSts; 	// Status of each Event State (0= OFF, 1=ON)
END_VAR
VAR
	{attribute 'OPC.UA.DA' := '0'}
	Conv_fbIntrlks				: FB_Intlks_Latch;
	Conv_IntlksArry				: ARRAY[0..15] OF BOOL;
	{attribute 'OPC.UA.DA' := '0'}
	Conv_fbEquipCntrl			: FB_EquipCntrl;
	{attribute 'OPC.UA.DA' := '0'}
	Conv_EventManager			: FB_EventMngr;
	Conv_CrrntExitPEJamDetctd	: FB_JamDetect;
	Conv_EventArry				: ARRAY[0..15] OF BOOL;
	
	Conv_LatchIgnore			: BOOL := FALSE;		// Put as a place holder for ease of future use
	Conv_LatchReset				: BOOL := FALSE;		//Put as a place holder for ease of future use
	Conv_IntlkBypassed			: ARRAY [0..15] OF BOOL;		//Put as a place holder for ease of future use
	Conv_RunEnabled				: BOOL;					// TRUE = Enable the conveyor to run
	Conv_StartEnabled			: BOOL;					// TRUE = Start Motion for Conv Enabled
	Conv_StartAllowed			: BOOL;					// TRUE = Start Motion for Conv Allowed

	// Sleep Timer
	fbSleepCntrl				: FB_SleepCntrl;

	// Start-up Delay Timer
	tStartUpDelay				: TON;

END_VAR

(*
	Depending on the conveyor type, the Interlock and Event 0 is different
	Also, jams are only detected on standard and end conveyors

	If no valid conveyor type is specified, the default is a standard type
*)

CASE Cfg_ConvType OF
	E_ConvType.standard:
		Conv_IntlksArry[0] := In_ConvDwnStrmMtrStatus OR (NOT In_ConvDwnStrmMtrStatus AND NOT In_ConvCrntExitPhotoEye);
		Conv_EventArry[0] := Conv_CrrntExitPEJamDetctd.JamDetected;
		Conv_CrrntExitPEJamDetctd(
			In_PE:= In_ConvCrntExitPhotoEye, 
			In_Status:= Out_ConvCrntMtr_Raw, 
			CFG_PEOKState:= 0, 
			JamDetTime:= cfg_JamDetectTime);
	E_ConvType.end:
		Conv_IntlksArry[0] := Conv_CrrntExitPEJamDetctd.JamDetected;
		Conv_EventArry[0] := In_EquipEvents.0;
		Conv_CrrntExitPEJamDetctd(
			In_PE:= In_ConvCrntExitPhotoEye, 
			In_Status:= Out_ConvCrntMtr_Raw, 
			CFG_PEOKState:= 0, 
			JamDetTime:= cfg_JamDetectTime);
	E_ConvType.slave:
		Conv_IntlksArry[0] := In_ConvDwnStrmMtrStatus;
		Conv_EventArry[0] := In_EquipEvents.0;
	ELSE
		Conv_IntlksArry[0] := In_ConvDwnStrmMtrStatus OR (NOT In_ConvDwnStrmMtrStatus AND NOT In_ConvCrntExitPhotoEye);
		Conv_EventArry[0] := Conv_CrrntExitPEJamDetctd.JamDetected;
		Conv_CrrntExitPEJamDetctd(
			In_PE:= In_ConvCrntExitPhotoEye, 
			In_Status:= Out_ConvCrntMtr_Raw, 
			CFG_PEOKState:= 0, 
			JamDetTime:= cfg_JamDetectTime);
END_CASE
// Set Up Common Converyor Interlocks and inputs for interlocks
Conv_IntlksArry[1] := System.SysIntlksAllOk; 
Conv_IntlksArry[2] := In_EquipIntlks.2;
Conv_IntlksArry[3] := In_EquipIntlks.3;
Conv_IntlksArry[4] := In_EquipIntlks.4;
Conv_IntlksArry[5] := In_EquipIntlks.5;
Conv_IntlksArry[6] := In_EquipIntlks.6;
Conv_IntlksArry[7] := In_EquipIntlks.7;
Conv_IntlksArry[8] := In_EquipIntlks.8;
Conv_IntlksArry[9] := In_EquipIntlks.9; 
Conv_IntlksArry[10] := In_EquipIntlks.10;
Conv_IntlksArry[11] := In_EquipIntlks.11;
Conv_IntlksArry[12] := In_EquipIntlks.12;
Conv_IntlksArry[13] := In_EquipIntlks.13;
Conv_IntlksArry[14] := In_EquipIntlks.14;
Conv_IntlksArry[15] := Conv_StartAllowed;
	
// Call Interlock block
Conv_fbIntrlks(
	In_Intlks:= Conv_IntlksArry,
	CFG_IntlksArry:= Cfg_EquipIntlksArry, 
	HMI_LatchIgnore:= Conv_LatchIgnore, 
	HMI_LatchReset:= Conv_LatchReset, 
	All_Intlk_OK=> Sts_EquipState.Sts_All_Intlks_OK, 
	STS_Intlks=> Sts_IntlksArry);
	
// Set Up Common Converyor Events and inputs for events
Conv_EventArry[1]:=	In_EquipEvents.1;
Conv_EventArry[2]:= In_EquipEvents.2;
Conv_EventArry[3]:= In_EquipEvents.3;
Conv_EventArry[4]:= In_EquipEvents.4;
Conv_EventArry[5]:= In_EquipEvents.5;
Conv_EventArry[6]:= In_EquipEvents.6;
Conv_EventArry[7]:= In_EquipEvents.7;
Conv_EventArry[8]:= In_EquipEvents.8;
Conv_EventArry[9]:= In_EquipEvents.9;
Conv_EventArry[10]:= In_EquipEvents.10;
Conv_EventArry[11]:= In_EquipEvents.11;
Conv_EventArry[12]:= In_EquipEvents.12;
Conv_EventArry[13]:= In_EquipEvents.13;
Conv_EventArry[14]:= In_EquipEvents.14;
Conv_EventArry[15]:= In_EquipEvents.15;

// Event Manager
Conv_EventManager(
	sEquipStateCntrlSts := Sts_EquipState.Sts_EquipmentState,
	In_EventsArry := Conv_EventArry ,  
	CFG_EvntsArry:= Cfg_EquipEvntsArry, 
	HMI_LatchReset:= In_o_EquipStatePB.ResetPB OR In_p_EquipStatePB.ResetPB,
	Out_FaultActive=> Sts_EquipState.Sts_FaultActive, 
	Out_WarnActive=> Sts_EquipState.Sts_WarnActive, 
	Sts_All_Evnts_OK=> Sts_EquipState.Sts_All_Evnts_OK, 
	Sts_FaultsArry=> Sts_FaultsArry, 
	Sts_WarnsArry=> Sts_WarnsArry, 
	Sts_EvntsArry=> Sts_EvntsArry);
	
//Call Equipment FB to control current motor	
Conv_fbEquipCntrl(
	CFG_EquipIndex := cfg_EquipIndex,
	CFG_EquipLabel := Cfg_EquipLabel,
	CFG_UseStrtCnd:= FALSE, 
	CFG_UseIntrlks:= TRUE, 
	CFG_UseHrnDly:= Cfg_UseStartUpDelay, 
	CFG_EquipDefState:= Cfg_EquipDefState, 
	In_IntlksOK:= Sts_EquipState.Sts_All_Intlks_OK, 
	In_SimActive:= In_SimActive, 
	In_Init:= In_EquipInit, 
	o_EquipStatePB:= In_o_EquipStatePB, 
	p_EquipStatePB:= In_p_EquipStatePB, 
	P_EquipReqRun:= In_P_ConvReqRun, 
	In_EquipFaults:= Sts_EquipState.Sts_FaultActive, 
	Out_EquipRun=> , 
	Out_Horn=> , 
	Sts_EquipState:= Sts_EquipState.Sts_EquipmentState);	

//===Sleep Timer
IF CFG_UseSleepTmr THEN
	fbSleepCntrl.In_Trigs.0 := In_ConvCrntExitPhotoEye OR In_p_EquipStatePB.AutoPB;
	fbSleepCntrl.In_Trigs.1 := In_WakeSlpTrigArry[1];
	fbSleepCntrl.In_Trigs.2 := In_WakeSlpTrigArry[2];
	fbSleepCntrl.In_Trigs.3 := In_WakeSlpTrigArry[3];
	fbSleepCntrl.In_Trigs.4 := In_WakeSlpTrigArry[4];
	fbSleepCntrl.In_Trigs.5 := In_WakeSlpTrigArry[5];
	fbSleepCntrl( 
		In_CrntFeedBack:= Out_ConvCrntMtr_Raw, 
		In_ConvState := Sts_EquipState.Sts_EquipmentState.CrntState,
		CFG_WaitToSlpTime:= Cfg_SleepWaitTime,
		SleepActive=> Sts_EquipState.Sts_SleepingActive);
ELSE
	Sts_EquipState.Sts_SleepingActive := FALSE;
END_IF
Sts_ConvSleepingActive := Sts_EquipState.Sts_SleepingActive;

(*
	Process the Conv_StartAllowed signal
	The Conv_StartAllowed enforces the cascade start of conveyors by waiting for the downstream motor to be running before
	this conveyor starts.
	Any conveyor can be started using the Start/Auto push-button without waiting for the downstream conveyor to be running.
*)
IF Sts_EquipState.Sts_EquipmentState.StsAuto THEN
	IF NOT Conv_StartAllowed THEN
		Conv_StartAllowed := In_ConvDwnStrmMtrStatus OR In_o_EquipStatePB.AutoPB OR (Cfg_ConvType = E_ConvType.end) OR (NOT Cfg_UseStartUpDelay);
	END_IF
ELSE
	Conv_StartAllowed := FALSE;
END_IF

// Process the Conv_RunEnabled signal
Conv_RunEnabled := Conv_fbEquipCntrl.Out_EquipRun
				AND NOT (Sts_EquipState.Sts_SleepingActive) 
				AND (Sts_EquipState.Sts_EquipmentState.StsMan OR (Sts_EquipState.Sts_EquipmentState.StsAuto AND Conv_StartAllowed));

// Use or do not use a start-up delay
IF Cfg_UseStartUpDelay THEN
	tStartUpDelay(IN := Conv_RunEnabled
					, PT := Cfg_StartUpDelayTime
					, Q =>);
	IF tStartUpDelay.Q THEN
		Conv_StartEnabled := TRUE;
	ELSE
		Conv_StartEnabled := FALSE;
	END_IF
ELSE
		Conv_StartEnabled := Conv_RunEnabled;	
END_IF

// Run motor based on the results of the Equipment Control and sleeping state
Out_ConvCrntMtr_Raw := Conv_StartEnabled;

// Capture WarnActive to carry these attributes into the Equipment state for System State reporting and display
Sts_EquipState.Sts_EquipmentState.StsHasWarnings := Sts_EquipState.Sts_WarnActive;

// Set Conveyor Motor Running Status
Sts_ConvCrntMtr := (CFG_UseMtrFdbck AND In_EquipMtrFdbck) OR (NOT CFG_UseMtrFdbck AND Out_ConvCrntMtr_Raw) OR (In_SimActive AND Conv_fbEquipCntrl.RunApproved);

// Capture the Operation state of the Conveyor
IF Sts_ConvCrntMtr THEN
	// Conveyor Running
	Sts_EquipState.Sts_EquipmentState.CrntOperState := E_OperStateCntrl.running;
ELSE
	IF Sts_EquipState.Sts_SleepingActive THEN
		// Conveyor Sleeping
		Sts_EquipState.Sts_EquipmentState.CrntOperState := E_OperStateCntrl.sleeping;
	ELSE
		// Conveyor Stopped
		Sts_EquipState.Sts_EquipmentState.CrntOperState := E_OperStateCntrl.stopped;
	END_IF
END_IF

//invert output
IF Cfg_InvertMotorOut THEN
    Out_ConvCrntMtr := NOT Out_ConvCrntMtr_Raw;
ELSE
    Out_ConvCrntMtr := Out_ConvCrntMtr_Raw;
END_IF

// Populate the Sts Output Variables
Sts_All_Intlks_OK  := Sts_EquipState.Sts_All_Intlks_OK;
Sts_All_Evnts_OK  := Sts_EquipState.Sts_All_Evnts_OK;
Sts_FaultActive := Sts_EquipState.Sts_FaultActive;
Sts_WarnActive := Sts_EquipState.Sts_WarnActive;

END_FUNCTION_BLOCK

// ---- POUs/System.TcPOU
PROGRAM System
VAR
	SysStateCntrlSts        	:    ST_EquipmentStatus;    // System State/Control/Status Data
    SysState                	:    FB_SystemCntrl;
    SysStateCntrl_StatePB       :    ST_StateCntrlPB;

    SysIntlksAllOk AT %Q*    	:    BOOL;    // Bit to show that System interlocks are OK   
    SysEventsAllOk AT %Q*		: 	BOOL;    // Bit to show that Syetem events are all OK If system events are needed use event manager FB tie to here
	
	ConvDefaultState AT %Q*		: 	E_StateCntrl := E_StateCntrl.stManual;	// The default state of all conveyors
	Sys_SimActive AT %Q*		: 	BOOL;	// Bit for simulation
	
	{attribute 'OPC.UA.DA' := '1'}
	HMI_PBSysStart:	BOOL;
	{attribute 'OPC.UA.DA' := '1'}
	HMI_PBSysStop:	BOOL;
	{attribute 'OPC.UA.DA' := '1'}
	HMI_PBSysReset:	BOOL;
	
	SysShrtPulseTmr: FB_Flasher;
	SysShrtPlsOnTime: TIME := T#750MS;
	SysShrtPlsOffTime: TIME := T#750MS;
	
	Cnvyr_Auto AT %Q*:	BOOL;		// Bit to send to all conveyors to put them in Auto mode
	Cnvyr_Manual AT %Q*:	BOOL;	// Bit to send to all conveyors to put them in Manual mode
	Cnvyr_Offline AT %Q*:	BOOL;	// Bit to send to all conveyors to put them in Offline mode -- Not used here
	Cnvyr_Reset AT %Q*:	BOOL;		// Bit to send to all conveyors to reset faults, safeties and etc

	Safety_Reset:	BOOL;
	tpSafetyReset:		TP := (PT := T#250MS);
	fSafetyReset:		F_TRIG;

	tpConvReset:		TP := (PT := T#250MS);
	
	ResetInit:	BOOL;	// Start the Safety/standard reset process

	Cnvyr_AlertTime:	TIME := T#5S;	
	Cnvyr_DelayTime:	TIME := T#1S;	
	Start_PulseWidth:	TIME := T#100MS;
	AlertDelay: FB_AlrtStrtDelay;
	
	nStatusArrayIndex : DINT;	// Increment to process the SysEquipStatusArray
	nTempStsIndex : DINT := 0;	// Used to Prevent Status Array Index duplicate assignments 

	ConveyorHasWarn: BOOL;
	ConveyorHasFault: BOOL;
	ConveyorIsSleeping: BOOL;
	ConveyorInAuto: BOOL;
	nTempRemoteIndex: DINT := 0;	//Temporary Remote Index to Simplify Code
	
END_VAR

VAR PERSISTENT    {attribute 'OPC.UA.DA' := '1'}
    cfgSysStateIntlksArry: ARRAY [0..15] OF ST_CfgEvents;
    {attribute 'OPC.UA.DA' := '1'}
    cfgSysStateEvntsArry: ARRAY [0..15] OF ST_CfgEvents;
END_VAR

// Send out reset PB put here in case added logic was needed
SysStateCntrl_StatePB.ResetPB := GVL_IO.PB_SysReset OR HMI_PBSysReset OR GVL_IO.PB_RemoteReset_12181 OR GVL_IO.PB_RemoteReset_7281; 
SysStateCntrl_StatePB.AutoPB := (HMI_PBSysStart OR GVL_IO.PB_SysStart) AND SysIntlksAllOk;
SysStateCntrl_StatePB.StopPB := HMI_PBSysStop OR (NOT GVL_IO.PB_SysStop);

// Set up system short pulse for alarm beacons, horns ets
SysShrtPulseTmr(In_Trig:= TRUE , Cfg_OnTime:= SysShrtPlsOnTime, Cfg_OffTime:= SysShrtPlsOffTime, Output=> );

// Set up System Interlocks

SysState.In_SystemIntlks.0 := GVL_IO.SystemAirPressure;
SysState.In_SystemIntlks.1 := SystemSafety.System_SafetyState.InRun;

// Setup the InterlockArray since persistent data items cannot by initilaized the same
(*
// Index 0
cfgSysStateIntlksArry[0].Description := 'System Air Pressure';
cfgSysStateIntlksArry[0].DeviceLabel := 'PS8222';
cfgSysStateIntlksArry[0].OKState := TRUE;
// Index 1
cfgSysStateIntlksArry[1].Description := ' Safety Running';
cfgSysStateIntlksArry[1].DeviceLabel := 'SYSTEM';
cfgSysStateIntlksArry[1].OKState := TRUE;
*)

// Set up System Events

SysState.In_SystemEvents.0 := GVL_IO.PanelEstop_OK;
SysState.In_SystemEvents.1 := GVL_IO.Remote_PullCord6040_OK;
SysState.In_SystemEvents.2 := GVL_IO.Remote_PullCord7004_OK;
SysState.In_SystemEvents.3 := SystemSafety.SecondFloorShaft_Estop_OK;
SysState.In_SystemEvents.4 := SystemSafety.ThirdFloorShaft_Estop_OK;
SysState.In_SystemEvents.5 := SystemSafety.System_SafetyState.CommErrAck;
SysState.In_SystemEvents.6 := SystemSafety.System_SafetyState.FBErr;
SysState.In_SystemEvents.7 := SystemSafety.System_SafetyState.OtherErr;

// Setup the EventArray since persistent data items cannot by initilaized the same
(*
// Index 0
cfgSysStateEvntsArry[0].Description := 'Panel E-Stop';
cfgSysStateEvntsArry[0].DeviceLabel := 'PB1';
cfgSysStateEvntsArry[0].OKState := TRUE;
cfgSysStateEvntsArry[0].StopCode := E_StopCodes.SystemStop;
// Index 1
cfgSysStateEvntsArry[1].Description := 'PullCord 6040';
cfgSysStateEvntsArry[1].DeviceLabel := 'P6040';
cfgSysStateEvntsArry[1].OKState := TRUE;
cfgSysStateEvntsArry[1].StopCode := E_StopCodes.SystemStop;
// Index 2
cfgSysStateEvntsArry[2].Description := 'PullCord 7004';
cfgSysStateEvntsArry[2].DeviceLabel := 'P7004';
cfgSysStateEvntsArry[2].OKState := TRUE;
cfgSysStateEvntsArry[2].StopCode := E_StopCodes.SystemStop;
// Index 3
cfgSysStateEvntsArry[3].Description := 'Second Floor Shaft EStop';
cfgSysStateEvntsArry[3].DeviceLabel := 'Shaft';
cfgSysStateEvntsArry[3].OKState := TRUE;
cfgSysStateEvntsArry[3].StopCode := E_StopCodes.SystemStop;
// Index 4
cfgSysStateEvntsArry[4].Description := 'Third Floor Shaft EStop';
cfgSysStateEvntsArry[4].DeviceLabel := 'Shaft';
cfgSysStateEvntsArry[4].OKState := TRUE;
cfgSysStateEvntsArry[4].StopCode := E_StopCodes.SystemStop;
// Index 5
cfgSysStateEvntsArry[5].Description := 'Safety Communication Error';
cfgSysStateEvntsArry[5].DeviceLabel := 'SYSTEM';
cfgSysStateEvntsArry[5].OKState := FALSE;
cfgSysStateEvntsArry[5].StopCode := E_StopCodes.SystemStop;
// Index 6
cfgSysStateEvntsArry[6].Description := 'Safety Function Block Error';
cfgSysStateEvntsArry[6].DeviceLabel := 'SYSTEM';
cfgSysStateEvntsArry[6].OKState := FALSE;
cfgSysStateEvntsArry[6].StopCode := E_StopCodes.SystemStop;
// Index 7
cfgSysStateEvntsArry[7].Description := 'Safety System Error';
cfgSysStateEvntsArry[7].DeviceLabel := 'SYSTEM';
cfgSysStateEvntsArry[7].OKState := FALSE;
cfgSysStateEvntsArry[7].StopCode := E_StopCodes.SystemStop;
*)
// Function Call
SysState(
    In_p_EquipStatePB:= SysStateCntrl_StatePB,
	Cfg_EquipLabel := '2nd Floor Totes',  
    Cfg_EquipIntlksArry:= cfgSysStateIntlksArry,
    Cfg_EquipEvntsArry:= cfgSysStateEvntsArry, 
    Sts_EquipState := SysStateCntrlSts,
	Out_Reset => ResetInit
);

SysIntlksAllOk := SysState.Sts_All_Intlks_OK;
SysEventsAllOk := SysState.Sts_All_Evnts_OK;

// Separate Standard/safety resets
tpSafetyReset(IN:= ResetInit);
// On While the timer is timing
Safety_Reset := tpSafetyReset.Q;

// On when the safety pulse goes low
fSafetyReset(CLK := tpSafetyReset.Q);
tpConvReset(IN := fSafetyReset.Q);
// On while the timer is timing
Cnvyr_Reset := tpConvReset.Q;

// Set up Start up delay and Auto/Manual control for conveyors

// Offline is set up in conveyors but has no logic here controlling it(This could be added here)
AlertDelay(
	In_StrtPulse:= SysState.Out_Auto , 
	In_StpPulse:= SysState.Out_Stop,
	CFG_AlertTime:= Cnvyr_AlertTime, 
	CFG_WaitTime:= Cnvyr_DelayTime,
	CFG_PulseTime:= Start_PulseWidth,
	In_ManTstTrig:= , 
	In_BypssDelay:= , 
	Out_Timed => Cnvyr_Auto,
	Out_Pulse => , 
	Out_Alert=> GVL_IO.HornMainPanel, 
	WaitActive=> );

Cnvyr_Manual:= SysState.Out_Stop; 	

//===========================================================================================
// Serialize the reporting equipment

// Set the value of System_Equip_Count, TempStsIndex should always match the number of identified statuses
GVL_EquipArrays.nSystemEquip_Count := nTempStsIndex;

// Control tower light
// Initialize the Equipment state detection
ConveyorHasWarn := 0;
ConveyorHasFault := 0;
ConveyorIsSleeping := 0;
ConveyorInAuto := 0;

//Conveyor Equipment
IF GVL_EquipArrays.nEquipIndex <> 0 THEN
    FOR nStatusArrayIndex := 1 TO GVL_EquipArrays.nEquipIndex BY 1 DO
        // Test for an already assigned Index value, but only to the outbound index, eventually this will populate the inbound value
        IF GVL_EquipArrays.aEquipStatusArray_Out[nStatusArrayIndex].RemIndex = 0 THEN
            // Increment the TempStsIndex only when we need to
            nTempStsIndex := nTempStsIndex + 1;
            // Assign the Remote Index to the Conveyor Status Data Item
            GVL_EquipArrays.aEquipStatusArray_Out[nStatusArrayIndex].RemIndex := nTempStsIndex;
        END_IF
        // Assign the Conveyor Status Value to the Status Array
        nTempRemoteIndex := GVL_EquipArrays.aEquipStatusArray_Out[nStatusArrayIndex].RemIndex;
        GVL_EquipArrays.aSystemEquipStatusArray[nTempRemoteIndex] := GVL_EquipArrays.aEquipStatusArray_In[nStatusArrayIndex];
    END_FOR
END_IF

// All System Equipment
IF GVL_EquipArrays.nSystemEquip_Count <> 0 THEN
	FOR nStatusArrayIndex := 1 TO GVL_EquipArrays.nSystemEquip_Count BY 1 DO
		// Only process the equipment if is is not in an offline state, this allows for the separate PLC equipment to 
		IF GVL_EquipArrays.aSystemEquipStatusArray[nStatusArrayIndex].CrntState <> E_StateCntrl.stOffline THEN
			// Test for an active warning on a coveyor
			IF GVL_EquipArrays.aSystemEquipStatusArray[nStatusArrayIndex].StsHasWarnings THEN
				ConveyorHasWarn := 1;
			END_IF
			// Test for an active Equipment fault, more than just a conveyor fault, could include Remote/IO, Barcode reader, etc..
			IF GVL_EquipArrays.aSystemEquipStatusArray[nStatusArrayIndex].StsFaulted THEN
				ConveyorHasFault := 1;
			END_IF
			// Test for a sleeping state
			IF GVL_EquipArrays.aSystemEquipStatusArray[nStatusArrayIndex].CrntOperState = E_OperStateCntrl.sleeping THEN
				ConveyorIsSleeping := 1;
			END_IF
			// Test for the Auto state, again an equipment state test to include non-conveyor equipment
			IF GVL_EquipArrays.aSystemEquipStatusArray[nStatusArrayIndex].StsAuto THEN
				ConveyorInAuto := 1;
			END_IF
		END_IF
	END_FOR
END_IF

// Initialise the Stack Light, only changing values as required
GVL_IO.LT_MainPanelStack_Green := FALSE;
GVL_IO.LT_MainPanelStack_Yellow := FALSE;
GVL_IO.LT_MainPanelStack_Red := FALSE;
	
IF ConveyorHasFault OR NOT SystemSafety.Safety_SystemEstopsOK THEN
	// Red light SOLID ON
	GVL_IO.LT_MainPanelStack_Red := TRUE;
ELSE
	IF ConveyorHasWarn THEN
		// Orange Light SOLID ON
		GVL_IO.LT_MainPanelStack_Yellow := TRUE;
	ELSE
		IF ConveyorInAuto THEN
			// Green Light SOLID ON
			GVL_IO.LT_MainPanelStack_Green := TRUE;
		ELSE
			GVL_IO.LT_MainPanelStack_Green := SysShrtPulseTmr.Output;
		END_IF
	END_IF
	IF GVL_IO.HornMainPanel THEN
		// Orange Light FLASHING ON
		GVL_IO.LT_MainPanelStack_Yellow := SysShrtPulseTmr.Output;
	END_IF;
END_IF

// Initialise the Stack Light, only changing values as required
GVL_IO.LT_7271_Green := FALSE;
GVL_IO.LT_7241_Yellow := FALSE;
GVL_IO.LT_7221_Red := FALSE;
	
